Fanuc TP program (LS listing): S004.LS

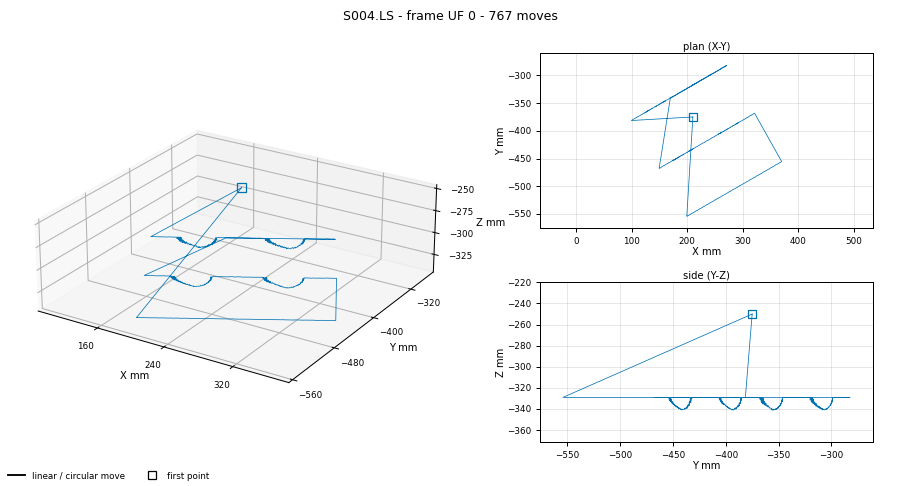
[picture p0: tool path of S004.LS in frame UF 0, 767 of 767 moves have a stored position in this frame; points joined in program order, loops and branches not executed]
/PROG  S004.LS
/ATTR
OWNER       = MNEDITOR;
COMMENT     = "";
PROG_SIZE   = 636;
CREATE      = DATE 23-01-07  TIME 11:59:14;
MODIFIED    = DATE 23-01-07  TIME 12:02:18;
FILE_NAME   = ;
VERSION     = 0;
LINE_COUNT  = 4;
MEMORY_SIZE = 992;
PROTECT     = READ_WRITE;
TCD:  STACK_SIZE	= 0,
      TASK_PRIORITY	= 50,
      TIME_SLICE	= 0,
      BUSY_LAMP_OFF	= 0,
      ABORT_REQUEST	= 0,
      PAUSE_REQUEST	= 0;
DEFAULT_GROUP	= 1,*,*,*,*;
CONTROL_CODE	= 00000000 00000000;
/MN
   1:J P[1] 100% FINE    ;
   2:L P[2] 100mm/sec CNT100    ;
   3:L P[3] 100mm/sec CNT100    ;
   4:L P[4] 100mm/sec CNT100    ;
   5:L P[5] 100mm/sec CNT100    ;
   6:L P[6] 100mm/sec CNT100    ;
   7:L P[7] 100mm/sec CNT100    ;
   8:L P[8] 100mm/sec CNT100    ;
   9:L P[9] 100mm/sec CNT100    ;
   10:L P[10] 100mm/sec CNT100    ;
   11:L P[11] 100mm/sec CNT100    ;
   12:L P[12] 100mm/sec CNT100    ;
   13:L P[13] 100mm/sec CNT100    ;
   14:L P[14] 100mm/sec CNT100    ;
   15:L P[15] 100mm/sec CNT100    ;
   16:L P[16] 100mm/sec CNT100    ;
   17:L P[17] 100mm/sec CNT100    ;
   18:L P[18] 100mm/sec CNT100    ;
   19:L P[19] 100mm/sec CNT100    ;
   20:L P[20] 100mm/sec CNT100    ;
   21:L P[21] 100mm/sec CNT100    ;
   22:L P[22] 100mm/sec CNT100    ;
   23:L P[23] 100mm/sec CNT100    ;
   24:L P[24] 100mm/sec CNT100    ;
   25:L P[25] 100mm/sec CNT100    ;
   26:L P[26] 100mm/sec CNT100    ;
   27:L P[27] 100mm/sec CNT100    ;
   28:L P[28] 100mm/sec CNT100    ;
   29:L P[29] 100mm/sec CNT100    ;
   30:L P[30] 100mm/sec CNT100    ;
   31:L P[31] 100mm/sec CNT100    ;
   32:L P[32] 100mm/sec CNT100    ;
   33:L P[33] 100mm/sec CNT100    ;
   34:L P[34] 100mm/sec CNT100    ;
   35:L P[35] 100mm/sec CNT100    ;
   36:L P[36] 100mm/sec CNT100    ;
   37:L P[37] 100mm/sec CNT100    ;
   38:L P[38] 100mm/sec CNT100    ;
   39:L P[39] 100mm/sec CNT100    ;
   40:L P[40] 100mm/sec CNT100    ;
   41:L P[41] 100mm/sec CNT100    ;
   42:L P[42] 100mm/sec CNT100    ;
   43:L P[43] 100mm/sec CNT100    ;
   44:L P[44] 100mm/sec CNT100    ;
   45:L P[45] 100mm/sec CNT100    ;
   46:L P[46] 100mm/sec CNT100    ;
   47:L P[47] 100mm/sec CNT100    ;
   48:L P[48] 100mm/sec CNT100    ;
   49:L P[49] 100mm/sec CNT100    ;
   50:L P[50] 100mm/sec CNT100    ;
   51:L P[51] 100mm/sec CNT100    ;
   52:L P[52] 100mm/sec CNT100    ;
   53:L P[53] 100mm/sec CNT100    ;
   54:L P[54] 100mm/sec CNT100    ;
   55:L P[55] 100mm/sec CNT100    ;
   56:L P[56] 100mm/sec CNT100    ;
   57:L P[57] 100mm/sec CNT100    ;
   58:L P[58] 100mm/sec CNT100    ;
   59:L P[59] 100mm/sec CNT100    ;
   60:L P[60] 100mm/sec CNT100    ;
   61:L P[61] 100mm/sec CNT100    ;
   62:L P[62] 100mm/sec CNT100    ;
   63:L P[63] 100mm/sec CNT100    ;
   64:L P[64] 100mm/sec CNT100    ;
   65:L P[65] 100mm/sec CNT100    ;
   66:L P[66] 100mm/sec CNT100    ;
   67:L P[67] 100mm/sec CNT100    ;
   68:L P[68] 100mm/sec CNT100    ;
   69:L P[69] 100mm/sec CNT100    ;
   70:L P[70] 100mm/sec CNT100    ;
   71:L P[71] 100mm/sec CNT100    ;
   72:L P[72] 100mm/sec CNT100    ;
   73:L P[73] 100mm/sec CNT100    ;
   74:L P[74] 100mm/sec CNT100    ;
   75:L P[75] 100mm/sec CNT100    ;
   76:L P[76] 100mm/sec CNT100    ;
   77:L P[77] 100mm/sec CNT100    ;
   78:L P[78] 100mm/sec CNT100    ;
   79:L P[79] 100mm/sec CNT100    ;
   80:L P[80] 100mm/sec CNT100    ;
   81:L P[81] 100mm/sec CNT100    ;
   82:L P[82] 100mm/sec CNT100    ;
   83:L P[83] 100mm/sec CNT100    ;
   84:L P[84] 100mm/sec CNT100    ;
   85:L P[85] 100mm/sec CNT100    ;
   86:L P[86] 100mm/sec CNT100    ;
   87:L P[87] 100mm/sec CNT100    ;
   88:L P[88] 100mm/sec CNT100    ;
   89:L P[89] 100mm/sec CNT100    ;
   90:L P[90] 100mm/sec CNT100    ;
   91:L P[91] 100mm/sec CNT100    ;
   92:L P[92] 100mm/sec CNT100    ;
   93:L P[93] 100mm/sec CNT100    ;
   94:L P[94] 100mm/sec CNT100    ;
   95:L P[95] 100mm/sec CNT100    ;
   96:L P[96] 100mm/sec CNT100    ;
   97:L P[97] 100mm/sec CNT100    ;
   98:L P[98] 100mm/sec CNT100    ;
   99:L P[99] 100mm/sec CNT100    ;
   100:L P[100] 100mm/sec CNT100    ;
   101:L P[101] 100mm/sec CNT100    ;
   102:L P[102] 100mm/sec CNT100    ;
   103:L P[103] 100mm/sec CNT100    ;
   104:L P[104] 100mm/sec CNT100    ;
   105:L P[105] 100mm/sec CNT100    ;
   106:L P[106] 100mm/sec CNT100    ;
   107:L P[107] 100mm/sec CNT100    ;
   108:L P[108] 100mm/sec CNT100    ;
   109:L P[109] 100mm/sec CNT100    ;
   110:L P[110] 100mm/sec CNT100    ;
   111:L P[111] 100mm/sec CNT100    ;
   112:L P[112] 100mm/sec CNT100    ;
   113:L P[113] 100mm/sec CNT100    ;
   114:L P[114] 100mm/sec CNT100    ;
   115:L P[115] 100mm/sec CNT100    ;
   116:L P[116] 100mm/sec CNT100    ;
   117:L P[117] 100mm/sec CNT100    ;
   118:L P[118] 100mm/sec CNT100    ;
   119:L P[119] 100mm/sec CNT100    ;
   120:L P[120] 100mm/sec CNT100    ;
   121:L P[121] 100mm/sec CNT100    ;
   122:L P[122] 100mm/sec CNT100    ;
   123:L P[123] 100mm/sec CNT100    ;
   124:L P[124] 100mm/sec CNT100    ;
   125:L P[125] 100mm/sec CNT100    ;
   126:L P[126] 100mm/sec CNT100    ;
   127:L P[127] 100mm/sec CNT100    ;
   128:L P[128] 100mm/sec CNT100    ;
   129:L P[129] 100mm/sec CNT100    ;
   130:L P[130] 100mm/sec CNT100    ;
   131:L P[131] 100mm/sec CNT100    ;
   132:L P[132] 100mm/sec CNT100    ;
   133:L P[133] 100mm/sec CNT100    ;
   134:L P[134] 100mm/sec CNT100    ;
   135:L P[135] 100mm/sec CNT100    ;
   136:L P[136] 100mm/sec CNT100    ;
   137:L P[137] 100mm/sec CNT100    ;
   138:L P[138] 100mm/sec CNT100    ;
   139:L P[139] 100mm/sec CNT100    ;
   140:L P[140] 100mm/sec CNT100    ;
   141:L P[141] 100mm/sec CNT100    ;
   142:L P[142] 100mm/sec CNT100    ;
   143:L P[143] 100mm/sec CNT100    ;
   144:L P[144] 100mm/sec CNT100    ;
   145:L P[145] 100mm/sec CNT100    ;
   146:L P[146] 100mm/sec CNT100    ;
   147:L P[147] 100mm/sec CNT100    ;
   148:L P[148] 100mm/sec CNT100    ;
   149:L P[149] 100mm/sec CNT100    ;
   150:L P[150] 100mm/sec CNT100    ;
   151:L P[151] 100mm/sec CNT100    ;
   152:L P[152] 100mm/sec CNT100    ;
   153:L P[153] 100mm/sec CNT100    ;
   154:L P[154] 100mm/sec CNT100    ;
   155:L P[155] 100mm/sec CNT100    ;
   156:L P[156] 100mm/sec CNT100    ;
   157:L P[157] 100mm/sec CNT100    ;
   158:L P[158] 100mm/sec CNT100    ;
   159:L P[159] 100mm/sec CNT100    ;
   160:L P[160] 100mm/sec CNT100    ;
   161:L P[161] 100mm/sec CNT100    ;
   162:L P[162] 100mm/sec CNT100    ;
   163:L P[163] 100mm/sec CNT100    ;
   164:L P[164] 100mm/sec CNT100    ;
   165:L P[165] 100mm/sec CNT100    ;
   166:L P[166] 100mm/sec CNT100    ;
   167:L P[167] 100mm/sec CNT100    ;
   168:L P[168] 100mm/sec CNT100    ;
   169:L P[169] 100mm/sec CNT100    ;
   170:L P[170] 100mm/sec CNT100    ;
   171:L P[171] 100mm/sec CNT100    ;
   172:L P[172] 100mm/sec CNT100    ;
   173:L P[173] 100mm/sec CNT100    ;
   174:L P[174] 100mm/sec CNT100    ;
   175:L P[175] 100mm/sec CNT100    ;
   176:L P[176] 100mm/sec CNT100    ;
   177:L P[177] 100mm/sec CNT100    ;
   178:L P[178] 100mm/sec CNT100    ;
   179:L P[179] 100mm/sec CNT100    ;
   180:L P[180] 100mm/sec CNT100    ;
   181:L P[181] 100mm/sec CNT100    ;
   182:L P[182] 100mm/sec CNT100    ;
   183:L P[183] 100mm/sec CNT100    ;
   184:L P[184] 100mm/sec CNT100    ;
   185:L P[185] 100mm/sec CNT100    ;
   186:L P[186] 100mm/sec CNT100    ;
   187:L P[187] 100mm/sec CNT100    ;
   188:L P[188] 100mm/sec CNT100    ;
   189:L P[189] 100mm/sec CNT100    ;
   190:L P[190] 100mm/sec CNT100    ;
   191:L P[191] 100mm/sec CNT100    ;
   192:L P[192] 100mm/sec CNT100    ;
   193:L P[193] 100mm/sec CNT100    ;
   194:L P[194] 100mm/sec CNT100    ;
   195:L P[195] 100mm/sec CNT100    ;
   196:L P[196] 100mm/sec CNT100    ;
   197:L P[197] 100mm/sec CNT100    ;
   198:L P[198] 100mm/sec CNT100    ;
   199:L P[199] 100mm/sec CNT100    ;
   200:L P[200] 100mm/sec CNT100    ;
   201:L P[201] 100mm/sec CNT100    ;
   202:L P[202] 100mm/sec CNT100    ;
   203:L P[203] 100mm/sec CNT100    ;
   204:L P[204] 100mm/sec CNT100    ;
   205:L P[205] 100mm/sec CNT100    ;
   206:L P[206] 100mm/sec CNT100    ;
   207:L P[207] 100mm/sec CNT100    ;
   208:L P[208] 100mm/sec CNT100    ;
   209:L P[209] 100mm/sec CNT100    ;
   210:L P[210] 100mm/sec CNT100    ;
   211:L P[211] 100mm/sec CNT100    ;
   212:L P[212] 100mm/sec CNT100    ;
   213:L P[213] 100mm/sec CNT100    ;
   214:L P[214] 100mm/sec CNT100    ;
   215:L P[215] 100mm/sec CNT100    ;
   216:L P[216] 100mm/sec CNT100    ;
   217:L P[217] 100mm/sec CNT100    ;
   218:L P[218] 100mm/sec CNT100    ;
   219:L P[219] 100mm/sec CNT100    ;
   220:L P[220] 100mm/sec CNT100    ;
   221:L P[221] 100mm/sec CNT100    ;
   222:L P[222] 100mm/sec CNT100    ;
   223:L P[223] 100mm/sec CNT100    ;
   224:L P[224] 100mm/sec CNT100    ;
   225:L P[225] 100mm/sec CNT100    ;
   226:L P[226] 100mm/sec CNT100    ;
   227:L P[227] 100mm/sec CNT100    ;
   228:L P[228] 100mm/sec CNT100    ;
   229:L P[229] 100mm/sec CNT100    ;
   230:L P[230] 100mm/sec CNT100    ;
   231:L P[231] 100mm/sec CNT100    ;
   232:L P[232] 100mm/sec CNT100    ;
   233:L P[233] 100mm/sec CNT100    ;
   234:L P[234] 100mm/sec CNT100    ;
   235:L P[235] 100mm/sec CNT100    ;
   236:L P[236] 100mm/sec CNT100    ;
   237:L P[237] 100mm/sec CNT100    ;
   238:L P[238] 100mm/sec CNT100    ;
   239:L P[239] 100mm/sec CNT100    ;
   240:L P[240] 100mm/sec CNT100    ;
   241:L P[241] 100mm/sec CNT100    ;
   242:L P[242] 100mm/sec CNT100    ;
   243:L P[243] 100mm/sec CNT100    ;
   244:L P[244] 100mm/sec CNT100    ;
   245:L P[245] 100mm/sec CNT100    ;
   246:L P[246] 100mm/sec CNT100    ;
   247:L P[247] 100mm/sec CNT100    ;
   248:L P[248] 100mm/sec CNT100    ;
   249:L P[249] 100mm/sec CNT100    ;
   250:L P[250] 100mm/sec CNT100    ;
   251:L P[251] 100mm/sec CNT100    ;
   252:L P[252] 100mm/sec CNT100    ;
   253:L P[253] 100mm/sec CNT100    ;
   254:L P[254] 100mm/sec CNT100    ;
   255:L P[255] 100mm/sec CNT100    ;
   256:L P[256] 100mm/sec CNT100    ;
   257:L P[257] 100mm/sec CNT100    ;
   258:L P[258] 100mm/sec CNT100    ;
   259:L P[259] 100mm/sec CNT100    ;
   260:L P[260] 100mm/sec CNT100    ;
   261:L P[261] 100mm/sec CNT100    ;
   262:L P[262] 100mm/sec CNT100    ;
   263:L P[263] 100mm/sec CNT100    ;
   264:L P[264] 100mm/sec CNT100    ;
   265:L P[265] 100mm/sec CNT100    ;
   266:L P[266] 100mm/sec CNT100    ;
   267:L P[267] 100mm/sec CNT100    ;
   268:L P[268] 100mm/sec CNT100    ;
   269:L P[269] 100mm/sec CNT100    ;
   270:L P[270] 100mm/sec CNT100    ;
   271:L P[271] 100mm/sec CNT100    ;
   272:L P[272] 100mm/sec CNT100    ;
   273:L P[273] 100mm/sec CNT100    ;
   274:L P[274] 100mm/sec CNT100    ;
   275:L P[275] 100mm/sec CNT100    ;
   276:L P[276] 100mm/sec CNT100    ;
   277:L P[277] 100mm/sec CNT100    ;
   278:L P[278] 100mm/sec CNT100    ;
   279:L P[279] 100mm/sec CNT100    ;
   280:L P[280] 100mm/sec CNT100    ;
   281:L P[281] 100mm/sec CNT100    ;
   282:L P[282] 100mm/sec CNT100    ;
   283:L P[283] 100mm/sec CNT100    ;
   284:L P[284] 100mm/sec CNT100    ;
   285:L P[285] 100mm/sec CNT100    ;
   286:L P[286] 100mm/sec CNT100    ;
   287:L P[287] 100mm/sec CNT100    ;
   288:L P[288] 100mm/sec CNT100    ;
   289:L P[289] 100mm/sec CNT100    ;
   290:L P[290] 100mm/sec CNT100    ;
   291:L P[291] 100mm/sec CNT100    ;
   292:L P[292] 100mm/sec CNT100    ;
   293:L P[293] 100mm/sec CNT100    ;
   294:L P[294] 100mm/sec CNT100    ;
   295:L P[295] 100mm/sec CNT100    ;
   296:L P[296] 100mm/sec CNT100    ;
   297:L P[297] 100mm/sec CNT100    ;
   298:L P[298] 100mm/sec CNT100    ;
   299:L P[299] 100mm/sec CNT100    ;
   300:L P[300] 100mm/sec CNT100    ;
   301:L P[301] 100mm/sec CNT100    ;
   302:L P[302] 100mm/sec CNT100    ;
   303:L P[303] 100mm/sec CNT100    ;
   304:L P[304] 100mm/sec CNT100    ;
   305:L P[305] 100mm/sec CNT100    ;
   306:L P[306] 100mm/sec CNT100    ;
   307:L P[307] 100mm/sec CNT100    ;
   308:L P[308] 100mm/sec CNT100    ;
   309:L P[309] 100mm/sec CNT100    ;
   310:L P[310] 100mm/sec CNT100    ;
   311:L P[311] 100mm/sec CNT100    ;
   312:L P[312] 100mm/sec CNT100    ;
   313:L P[313] 100mm/sec CNT100    ;
   314:L P[314] 100mm/sec CNT100    ;
   315:L P[315] 100mm/sec CNT100    ;
   316:L P[316] 100mm/sec CNT100    ;
   317:L P[317] 100mm/sec CNT100    ;
   318:L P[318] 100mm/sec CNT100    ;
   319:L P[319] 100mm/sec CNT100    ;
   320:L P[320] 100mm/sec CNT100    ;
   321:L P[321] 100mm/sec CNT100    ;
   322:L P[322] 100mm/sec CNT100    ;
   323:L P[323] 100mm/sec CNT100    ;
   324:L P[324] 100mm/sec CNT100    ;
   325:L P[325] 100mm/sec CNT100    ;
   326:L P[326] 100mm/sec CNT100    ;
   327:L P[327] 100mm/sec CNT100    ;
   328:L P[328] 100mm/sec CNT100    ;
   329:L P[329] 100mm/sec CNT100    ;
   330:L P[330] 100mm/sec CNT100    ;
   331:L P[331] 100mm/sec CNT100    ;
   332:L P[332] 100mm/sec CNT100    ;
   333:L P[333] 100mm/sec CNT100    ;
   334:L P[334] 100mm/sec CNT100    ;
   335:L P[335] 100mm/sec CNT100    ;
   336:L P[336] 100mm/sec CNT100    ;
   337:L P[337] 100mm/sec CNT100    ;
   338:L P[338] 100mm/sec CNT100    ;
   339:L P[339] 100mm/sec CNT100    ;
   340:L P[340] 100mm/sec CNT100    ;
   341:L P[341] 100mm/sec CNT100    ;
   342:L P[342] 100mm/sec CNT100    ;
   343:L P[343] 100mm/sec CNT100    ;
   344:L P[344] 100mm/sec CNT100    ;
   345:L P[345] 100mm/sec CNT100    ;
   346:L P[346] 100mm/sec CNT100    ;
   347:L P[347] 100mm/sec CNT100    ;
   348:L P[348] 100mm/sec CNT100    ;
   349:L P[349] 100mm/sec CNT100    ;
   350:L P[350] 100mm/sec CNT100    ;
   351:L P[351] 100mm/sec CNT100    ;
   352:L P[352] 100mm/sec CNT100    ;
   353:L P[353] 100mm/sec CNT100    ;
   354:L P[354] 100mm/sec CNT100    ;
   355:L P[355] 100mm/sec CNT100    ;
   356:L P[356] 100mm/sec CNT100    ;
   357:L P[357] 100mm/sec CNT100    ;
   358:L P[358] 100mm/sec CNT100    ;
   359:L P[359] 100mm/sec CNT100    ;
   360:L P[360] 100mm/sec CNT100    ;
   361:L P[361] 100mm/sec CNT100    ;
   362:L P[362] 100mm/sec CNT100    ;
   363:L P[363] 100mm/sec CNT100    ;
   364:L P[364] 100mm/sec CNT100    ;
   365:L P[365] 100mm/sec CNT100    ;
   366:L P[366] 100mm/sec CNT100    ;
   367:L P[367] 100mm/sec CNT100    ;
   368:L P[368] 100mm/sec CNT100    ;
   369:L P[369] 100mm/sec CNT100    ;
   370:L P[370] 100mm/sec CNT100    ;
   371:L P[371] 100mm/sec CNT100    ;
   372:L P[372] 100mm/sec CNT100    ;
   373:L P[373] 100mm/sec CNT100    ;
   374:L P[374] 100mm/sec CNT100    ;
   375:L P[375] 100mm/sec CNT100    ;
   376:L P[376] 100mm/sec CNT100    ;
   377:L P[377] 100mm/sec CNT100    ;
   378:L P[378] 100mm/sec CNT100    ;
   379:L P[379] 100mm/sec CNT100    ;
   380:L P[380] 100mm/sec CNT100    ;
   381:L P[381] 100mm/sec CNT100    ;
   382:L P[382] 100mm/sec CNT100    ;
   383:L P[383] 100mm/sec CNT100    ;
   384:L P[384] 100mm/sec CNT100    ;
   385:L P[385] 100mm/sec CNT100    ;
   386:L P[386] 100mm/sec CNT100    ;
   387:L P[387] 100mm/sec CNT100    ;
   388:L P[388] 100mm/sec CNT100    ;
   389:L P[389] 100mm/sec CNT100    ;
   390:L P[390] 100mm/sec CNT100    ;
   391:L P[391] 100mm/sec CNT100    ;
   392:L P[392] 100mm/sec CNT100    ;
   393:L P[393] 100mm/sec CNT100    ;
   394:L P[394] 100mm/sec CNT100    ;
   395:L P[395] 100mm/sec CNT100    ;
   396:L P[396] 100mm/sec CNT100    ;
   397:L P[397] 100mm/sec CNT100    ;
   398:L P[398] 100mm/sec CNT100    ;
   399:L P[399] 100mm/sec CNT100    ;
   400:L P[400] 100mm/sec CNT100    ;
   401:L P[401] 100mm/sec CNT100    ;
   402:L P[402] 100mm/sec CNT100    ;
   403:L P[403] 100mm/sec CNT100    ;
   404:L P[404] 100mm/sec CNT100    ;
   405:L P[405] 100mm/sec CNT100    ;
   406:L P[406] 100mm/sec CNT100    ;
   407:L P[407] 100mm/sec CNT100    ;
   408:L P[408] 100mm/sec CNT100    ;
   409:L P[409] 100mm/sec CNT100    ;
   410:L P[410] 100mm/sec CNT100    ;
   411:L P[411] 100mm/sec CNT100    ;
   412:L P[412] 100mm/sec CNT100    ;
   413:L P[413] 100mm/sec CNT100    ;
   414:L P[414] 100mm/sec CNT100    ;
   415:L P[415] 100mm/sec CNT100    ;
   416:L P[416] 100mm/sec CNT100    ;
   417:L P[417] 100mm/sec CNT100    ;
   418:L P[418] 100mm/sec CNT100    ;
   419:L P[419] 100mm/sec CNT100    ;
   420:L P[420] 100mm/sec CNT100    ;
   421:L P[421] 100mm/sec CNT100    ;
   422:L P[422] 100mm/sec CNT100    ;
   423:L P[423] 100mm/sec CNT100    ;
   424:L P[424] 100mm/sec CNT100    ;
   425:L P[425] 100mm/sec CNT100    ;
   426:L P[426] 100mm/sec CNT100    ;
   427:L P[427] 100mm/sec CNT100    ;
   428:L P[428] 100mm/sec CNT100    ;
   429:L P[429] 100mm/sec CNT100    ;
   430:L P[430] 100mm/sec CNT100    ;
   431:L P[431] 100mm/sec CNT100    ;
   432:L P[432] 100mm/sec CNT100    ;
   433:L P[433] 100mm/sec CNT100    ;
   434:L P[434] 100mm/sec CNT100    ;
   435:L P[435] 100mm/sec CNT100    ;
   436:L P[436] 100mm/sec CNT100    ;
   437:L P[437] 100mm/sec CNT100    ;
   438:L P[438] 100mm/sec CNT100    ;
   439:L P[439] 100mm/sec CNT100    ;
   440:L P[440] 100mm/sec CNT100    ;
   441:L P[441] 100mm/sec CNT100    ;
   442:L P[442] 100mm/sec CNT100    ;
   443:L P[443] 100mm/sec CNT100    ;
   444:L P[444] 100mm/sec CNT100    ;
   445:L P[445] 100mm/sec CNT100    ;
   446:L P[446] 100mm/sec CNT100    ;
   447:L P[447] 100mm/sec CNT100    ;
   448:L P[448] 100mm/sec CNT100    ;
   449:L P[449] 100mm/sec CNT100    ;
   450:L P[450] 100mm/sec CNT100    ;
   451:L P[451] 100mm/sec CNT100    ;
   452:L P[452] 100mm/sec CNT100    ;
   453:L P[453] 100mm/sec CNT100    ;
   454:L P[454] 100mm/sec CNT100    ;
   455:L P[455] 100mm/sec CNT100    ;
   456:L P[456] 100mm/sec CNT100    ;
   457:L P[457] 100mm/sec CNT100    ;
   458:L P[458] 100mm/sec CNT100    ;
   459:L P[459] 100mm/sec CNT100    ;
   460:L P[460] 100mm/sec CNT100    ;
   461:L P[461] 100mm/sec CNT100    ;
   462:L P[462] 100mm/sec CNT100    ;
   463:L P[463] 100mm/sec CNT100    ;
   464:L P[464] 100mm/sec CNT100    ;
   465:L P[465] 100mm/sec CNT100    ;
   466:L P[466] 100mm/sec CNT100    ;
   467:L P[467] 100mm/sec CNT100    ;
   468:L P[468] 100mm/sec CNT100    ;
   469:L P[469] 100mm/sec CNT100    ;
   470:L P[470] 100mm/sec CNT100    ;
   471:L P[471] 100mm/sec CNT100    ;
   472:L P[472] 100mm/sec CNT100    ;
   473:L P[473] 100mm/sec CNT100    ;
   474:L P[474] 100mm/sec CNT100    ;
   475:L P[475] 100mm/sec CNT100    ;
   476:L P[476] 100mm/sec CNT100    ;
   477:L P[477] 100mm/sec CNT100    ;
   478:L P[478] 100mm/sec CNT100    ;
   479:L P[479] 100mm/sec CNT100    ;
   480:L P[480] 100mm/sec CNT100    ;
   481:L P[481] 100mm/sec CNT100    ;
   482:L P[482] 100mm/sec CNT100    ;
   483:L P[483] 100mm/sec CNT100    ;
   484:L P[484] 100mm/sec CNT100    ;
   485:L P[485] 100mm/sec CNT100    ;
   486:L P[486] 100mm/sec CNT100    ;
   487:L P[487] 100mm/sec CNT100    ;
   488:L P[488] 100mm/sec CNT100    ;
   489:L P[489] 100mm/sec CNT100    ;
   490:L P[490] 100mm/sec CNT100    ;
   491:L P[491] 100mm/sec CNT100    ;
   492:L P[492] 100mm/sec CNT100    ;
   493:L P[493] 100mm/sec CNT100    ;
   494:L P[494] 100mm/sec CNT100    ;
   495:L P[495] 100mm/sec CNT100    ;
   496:L P[496] 100mm/sec CNT100    ;
   497:L P[497] 100mm/sec CNT100    ;
   498:L P[498] 100mm/sec CNT100    ;
   499:L P[499] 100mm/sec CNT100    ;
   500:L P[500] 100mm/sec CNT100    ;
   501:L P[501] 100mm/sec CNT100    ;
   502:L P[502] 100mm/sec CNT100    ;
   503:L P[503] 100mm/sec CNT100    ;
   504:L P[504] 100mm/sec CNT100    ;
   505:L P[505] 100mm/sec CNT100    ;
   506:L P[506] 100mm/sec CNT100    ;
   507:L P[507] 100mm/sec CNT100    ;
   508:L P[508] 100mm/sec CNT100    ;
   509:L P[509] 100mm/sec CNT100    ;
   510:L P[510] 100mm/sec CNT100    ;
   511:L P[511] 100mm/sec CNT100    ;
   512:L P[512] 100mm/sec CNT100    ;
   513:L P[513] 100mm/sec CNT100    ;
   514:L P[514] 100mm/sec CNT100    ;
   515:L P[515] 100mm/sec CNT100    ;
   516:L P[516] 100mm/sec CNT100    ;
   517:L P[517] 100mm/sec CNT100    ;
   518:L P[518] 100mm/sec CNT100    ;
   519:L P[519] 100mm/sec CNT100    ;
   520:L P[520] 100mm/sec CNT100    ;
   521:L P[521] 100mm/sec CNT100    ;
   522:L P[522] 100mm/sec CNT100    ;
   523:L P[523] 100mm/sec CNT100    ;
   524:L P[524] 100mm/sec CNT100    ;
   525:L P[525] 100mm/sec CNT100    ;
   526:L P[526] 100mm/sec CNT100    ;
   527:L P[527] 100mm/sec CNT100    ;
   528:L P[528] 100mm/sec CNT100    ;
   529:L P[529] 100mm/sec CNT100    ;
   530:L P[530] 100mm/sec CNT100    ;
   531:L P[531] 100mm/sec CNT100    ;
   532:L P[532] 100mm/sec CNT100    ;
   533:L P[533] 100mm/sec CNT100    ;
   534:L P[534] 100mm/sec CNT100    ;
   535:L P[535] 100mm/sec CNT100    ;
   536:L P[536] 100mm/sec CNT100    ;
   537:L P[537] 100mm/sec CNT100    ;
   538:L P[538] 100mm/sec CNT100    ;
   539:L P[539] 100mm/sec CNT100    ;
   540:L P[540] 100mm/sec CNT100    ;
   541:L P[541] 100mm/sec CNT100    ;
   542:L P[542] 100mm/sec CNT100    ;
   543:L P[543] 100mm/sec CNT100    ;
   544:L P[544] 100mm/sec CNT100    ;
   545:L P[545] 100mm/sec CNT100    ;
   546:L P[546] 100mm/sec CNT100    ;
   547:L P[547] 100mm/sec CNT100    ;
   548:L P[548] 100mm/sec CNT100    ;
   549:L P[549] 100mm/sec CNT100    ;
   550:L P[550] 100mm/sec CNT100    ;
   551:L P[551] 100mm/sec CNT100    ;
   552:L P[552] 100mm/sec CNT100    ;
   553:L P[553] 100mm/sec CNT100    ;
   554:L P[554] 100mm/sec CNT100    ;
   555:L P[555] 100mm/sec CNT100    ;
   556:L P[556] 100mm/sec CNT100    ;
   557:L P[557] 100mm/sec CNT100    ;
   558:L P[558] 100mm/sec CNT100    ;
   559:L P[559] 100mm/sec CNT100    ;
   560:L P[560] 100mm/sec CNT100    ;
   561:L P[561] 100mm/sec CNT100    ;
   562:L P[562] 100mm/sec CNT100    ;
   563:L P[563] 100mm/sec CNT100    ;
   564:L P[564] 100mm/sec CNT100    ;
   565:L P[565] 100mm/sec CNT100    ;
   566:L P[566] 100mm/sec CNT100    ;
   567:L P[567] 100mm/sec CNT100    ;
   568:L P[568] 100mm/sec CNT100    ;
   569:L P[569] 100mm/sec CNT100    ;
   570:L P[570] 100mm/sec CNT100    ;
   571:L P[571] 100mm/sec CNT100    ;
   572:L P[572] 100mm/sec CNT100    ;
   573:L P[573] 100mm/sec CNT100    ;
   574:L P[574] 100mm/sec CNT100    ;
   575:L P[575] 100mm/sec CNT100    ;
   576:L P[576] 100mm/sec CNT100    ;
   577:L P[577] 100mm/sec CNT100    ;
   578:L P[578] 100mm/sec CNT100    ;
   579:L P[579] 100mm/sec CNT100    ;
   580:L P[580] 100mm/sec CNT100    ;
   581:L P[581] 100mm/sec CNT100    ;
   582:L P[582] 100mm/sec CNT100    ;
   583:L P[583] 100mm/sec CNT100    ;
   584:L P[584] 100mm/sec CNT100    ;
   585:L P[585] 100mm/sec CNT100    ;
   586:L P[586] 100mm/sec CNT100    ;
   587:L P[587] 100mm/sec CNT100    ;
   588:L P[588] 100mm/sec CNT100    ;
   589:L P[589] 100mm/sec CNT100    ;
   590:L P[590] 100mm/sec CNT100    ;
   591:L P[591] 100mm/sec CNT100    ;
   592:L P[592] 100mm/sec CNT100    ;
   593:L P[593] 100mm/sec CNT100    ;
   594:L P[594] 100mm/sec CNT100    ;
   595:L P[595] 100mm/sec CNT100    ;
   596:L P[596] 100mm/sec CNT100    ;
   597:L P[597] 100mm/sec CNT100    ;
   598:L P[598] 100mm/sec CNT100    ;
   599:L P[599] 100mm/sec CNT100    ;
   600:L P[600] 100mm/sec CNT100    ;
   601:L P[601] 100mm/sec CNT100    ;
   602:L P[602] 100mm/sec CNT100    ;
   603:L P[603] 100mm/sec CNT100    ;
   604:L P[604] 100mm/sec CNT100    ;
   605:L P[605] 100mm/sec CNT100    ;
   606:L P[606] 100mm/sec CNT100    ;
   607:L P[607] 100mm/sec CNT100    ;
   608:L P[608] 100mm/sec CNT100    ;
   609:L P[609] 100mm/sec CNT100    ;
   610:L P[610] 100mm/sec CNT100    ;
   611:L P[611] 100mm/sec CNT100    ;
   612:L P[612] 100mm/sec CNT100    ;
   613:L P[613] 100mm/sec CNT100    ;
   614:L P[614] 100mm/sec CNT100    ;
   615:L P[615] 100mm/sec CNT100    ;
   616:L P[616] 100mm/sec CNT100    ;
   617:L P[617] 100mm/sec CNT100    ;
   618:L P[618] 100mm/sec CNT100    ;
   619:L P[619] 100mm/sec CNT100    ;
   620:L P[620] 100mm/sec CNT100    ;
   621:L P[621] 100mm/sec CNT100    ;
   622:L P[622] 100mm/sec CNT100    ;
   623:L P[623] 100mm/sec CNT100    ;
   624:L P[624] 100mm/sec CNT100    ;
   625:L P[625] 100mm/sec CNT100    ;
   626:L P[626] 100mm/sec CNT100    ;
   627:L P[627] 100mm/sec CNT100    ;
   628:L P[628] 100mm/sec CNT100    ;
   629:L P[629] 100mm/sec CNT100    ;
   630:L P[630] 100mm/sec CNT100    ;
   631:L P[631] 100mm/sec CNT100    ;
   632:L P[632] 100mm/sec CNT100    ;
   633:L P[633] 100mm/sec CNT100    ;
   634:L P[634] 100mm/sec CNT100    ;
   635:L P[635] 100mm/sec CNT100    ;
   636:L P[636] 100mm/sec CNT100    ;
   637:L P[637] 100mm/sec CNT100    ;
   638:L P[638] 100mm/sec CNT100    ;
   639:L P[639] 100mm/sec CNT100    ;
   640:L P[640] 100mm/sec CNT100    ;
   641:L P[641] 100mm/sec CNT100    ;
   642:L P[642] 100mm/sec CNT100    ;
   643:L P[643] 100mm/sec CNT100    ;
   644:L P[644] 100mm/sec CNT100    ;
   645:L P[645] 100mm/sec CNT100    ;
   646:L P[646] 100mm/sec CNT100    ;
   647:L P[647] 100mm/sec CNT100    ;
   648:L P[648] 100mm/sec CNT100    ;
   649:L P[649] 100mm/sec CNT100    ;
   650:L P[650] 100mm/sec CNT100    ;
   651:L P[651] 100mm/sec CNT100    ;
   652:L P[652] 100mm/sec CNT100    ;
   653:L P[653] 100mm/sec CNT100    ;
   654:L P[654] 100mm/sec CNT100    ;
   655:L P[655] 100mm/sec CNT100    ;
   656:L P[656] 100mm/sec CNT100    ;
   657:L P[657] 100mm/sec CNT100    ;
   658:L P[658] 100mm/sec CNT100    ;
   659:L P[659] 100mm/sec CNT100    ;
   660:L P[660] 100mm/sec CNT100    ;
   661:L P[661] 100mm/sec CNT100    ;
   662:L P[662] 100mm/sec CNT100    ;
   663:L P[663] 100mm/sec CNT100    ;
   664:L P[664] 100mm/sec CNT100    ;
   665:L P[665] 100mm/sec CNT100    ;
   666:L P[666] 100mm/sec CNT100    ;
   667:L P[667] 100mm/sec CNT100    ;
   668:L P[668] 100mm/sec CNT100    ;
   669:L P[669] 100mm/sec CNT100    ;
   670:L P[670] 100mm/sec CNT100    ;
   671:L P[671] 100mm/sec CNT100    ;
   672:L P[672] 100mm/sec CNT100    ;
   673:L P[673] 100mm/sec CNT100    ;
   674:L P[674] 100mm/sec CNT100    ;
   675:L P[675] 100mm/sec CNT100    ;
   676:L P[676] 100mm/sec CNT100    ;
   677:L P[677] 100mm/sec CNT100    ;
   678:L P[678] 100mm/sec CNT100    ;
   679:L P[679] 100mm/sec CNT100    ;
   680:L P[680] 100mm/sec CNT100    ;
   681:L P[681] 100mm/sec CNT100    ;
   682:L P[682] 100mm/sec CNT100    ;
   683:L P[683] 100mm/sec CNT100    ;
   684:L P[684] 100mm/sec CNT100    ;
   685:L P[685] 100mm/sec CNT100    ;
   686:L P[686] 100mm/sec CNT100    ;
   687:L P[687] 100mm/sec CNT100    ;
   688:L P[688] 100mm/sec CNT100    ;
   689:L P[689] 100mm/sec CNT100    ;
   690:L P[690] 100mm/sec CNT100    ;
   691:L P[691] 100mm/sec CNT100    ;
   692:L P[692] 100mm/sec CNT100    ;
   693:L P[693] 100mm/sec CNT100    ;
   694:L P[694] 100mm/sec CNT100    ;
   695:L P[695] 100mm/sec CNT100    ;
   696:L P[696] 100mm/sec CNT100    ;
   697:L P[697] 100mm/sec CNT100    ;
   698:L P[698] 100mm/sec CNT100    ;
   699:L P[699] 100mm/sec CNT100    ;
   700:L P[700] 100mm/sec CNT100    ;
   701:L P[701] 100mm/sec CNT100    ;
   702:L P[702] 100mm/sec CNT100    ;
   703:L P[703] 100mm/sec CNT100    ;
   704:L P[704] 100mm/sec CNT100    ;
   705:L P[705] 100mm/sec CNT100    ;
   706:L P[706] 100mm/sec CNT100    ;
   707:L P[707] 100mm/sec CNT100    ;
   708:L P[708] 100mm/sec CNT100    ;
   709:L P[709] 100mm/sec CNT100    ;
   710:L P[710] 100mm/sec CNT100    ;
   711:L P[711] 100mm/sec CNT100    ;
   712:L P[712] 100mm/sec CNT100    ;
   713:L P[713] 100mm/sec CNT100    ;
   714:L P[714] 100mm/sec CNT100    ;
   715:L P[715] 100mm/sec CNT100    ;
   716:L P[716] 100mm/sec CNT100    ;
   717:L P[717] 100mm/sec CNT100    ;
   718:L P[718] 100mm/sec CNT100    ;
   719:L P[719] 100mm/sec CNT100    ;
   720:L P[720] 100mm/sec CNT100    ;
   721:L P[721] 100mm/sec CNT100    ;
   722:L P[722] 100mm/sec CNT100    ;
   723:L P[723] 100mm/sec CNT100    ;
   724:L P[724] 100mm/sec CNT100    ;
   725:L P[725] 100mm/sec CNT100    ;
   726:L P[726] 100mm/sec CNT100    ;
   727:L P[727] 100mm/sec CNT100    ;
   728:L P[728] 100mm/sec CNT100    ;
   729:L P[729] 100mm/sec CNT100    ;
   730:L P[730] 100mm/sec CNT100    ;
   731:L P[731] 100mm/sec CNT100    ;
   732:L P[732] 100mm/sec CNT100    ;
   733:L P[733] 100mm/sec CNT100    ;
   734:L P[734] 100mm/sec CNT100    ;
   735:L P[735] 100mm/sec CNT100    ;
   736:L P[736] 100mm/sec CNT100    ;
   737:L P[737] 100mm/sec CNT100    ;
   738:L P[738] 100mm/sec CNT100    ;
   739:L P[739] 100mm/sec CNT100    ;
   740:L P[740] 100mm/sec CNT100    ;
   741:L P[741] 100mm/sec CNT100    ;
   742:L P[742] 100mm/sec CNT100    ;
   743:L P[743] 100mm/sec CNT100    ;
   744:L P[744] 100mm/sec CNT100    ;
   745:L P[745] 100mm/sec CNT100    ;
   746:L P[746] 100mm/sec CNT100    ;
   747:L P[747] 100mm/sec CNT100    ;
   748:L P[748] 100mm/sec CNT100    ;
   749:L P[749] 100mm/sec CNT100    ;
   750:L P[750] 100mm/sec CNT100    ;
   751:L P[751] 100mm/sec CNT100    ;
   752:L P[752] 100mm/sec CNT100    ;
   753:L P[753] 100mm/sec CNT100    ;
   754:L P[754] 100mm/sec CNT100    ;
   755:L P[755] 100mm/sec CNT100    ;
   756:L P[756] 100mm/sec CNT100    ;
   757:L P[757] 100mm/sec CNT100    ;
   758:L P[758] 100mm/sec CNT100    ;
   759:L P[759] 100mm/sec CNT100    ;
   760:L P[760] 100mm/sec CNT100    ;
   761:L P[761] 100mm/sec CNT100    ;
   762:L P[762] 100mm/sec CNT100    ;
   763:L P[763] 100mm/sec CNT100    ;
   764:L P[764] 100mm/sec CNT100    ;
   765:L P[765] 100mm/sec CNT100    ;
   766:L P[766] 100mm/sec CNT100    ;
   767:L P[767] 100mm/sec CNT100    ;
/POS
P[1]{
   GP1:
	UF : 0, UT : 6,		CONFIG : 'N U T, 0, 0, 0',
	X =  210.000  mm,	Y =   -375.000  mm,	Z =   -250.000  mm,
	W =  90.000 deg,	P =   0.000 deg,	R =   90.000 deg
};
P[2]{
   GP1:
	UF : 0, UT : 6,		CONFIG : 'N U T, 0, 0, 0',
	X =  99.048  mm,	Y =   -381.442  mm,	Z =   -329.000  mm,
	W =  90.000 deg,	P =   0.000 deg,	R =   90.000 deg
};
P[3]{
   GP1:
	UF : 0, UT : 6,		CONFIG : 'N U T, 0, 0, 0',
	X =  99.873  mm,	Y =   -380.917  mm,	Z =   -329.000  mm,
	W =  90.000 deg,	P =   0.000 deg,	R =   90.000 deg
};
P[4]{
   GP1:
	UF : 0, UT : 6,		CONFIG : 'N U T, 0, 0, 0',
	X =  100.888  mm,	Y =   -380.459  mm,	Z =   -329.000  mm,
	W =  90.000 deg,	P =   0.000 deg,	R =   90.000 deg
};
P[5]{
   GP1:
	UF : 0, UT : 6,		CONFIG : 'N U T, 0, 0, 0',
	X =  101.765  mm,	Y =   -379.889  mm,	Z =   -329.000  mm,
	W =  90.000 deg,	P =   0.000 deg,	R =   90.000 deg
};
P[6]{
   GP1:
	UF : 0, UT : 6,		CONFIG : 'N U T, 0, 0, 0',
	X =  102.835  mm,	Y =   -379.243  mm,	Z =   -329.000  mm,
	W =  90.000 deg,	P =   0.000 deg,	R =   90.000 deg
};
P[7]{
   GP1:
	UF : 0, UT : 6,		CONFIG : 'N U T, 0, 0, 0',
	X =  103.446  mm,	Y =   -378.703  mm,	Z =   -329.000  mm,
	W =  90.000 deg,	P =   0.000 deg,	R =   90.000 deg
};
P[8]{
   GP1:
	UF : 0, UT : 6,		CONFIG : 'N U T, 0, 0, 0',
	X =  104.720  mm,	Y =   -378.117  mm,	Z =   -329.100  mm,
	W =  90.000 deg,	P =   0.000 deg,	R =   90.000 deg
};
P[9]{
   GP1:
	UF : 0, UT : 6,		CONFIG : 'N U T, 0, 0, 0',
	X =  105.487  mm,	Y =   -377.698  mm,	Z =   -329.100  mm,
	W =  90.000 deg,	P =   0.000 deg,	R =   90.000 deg
};
P[10]{
   GP1:
	UF : 0, UT : 6,		CONFIG : 'N U T, 0, 0, 0',
	X =  106.013  mm,	Y =   -376.984  mm,	Z =   -329.100  mm,
	W =  90.000 deg,	P =   0.000 deg,	R =   90.000 deg
};
P[11]{
   GP1:
	UF : 0, UT : 6,		CONFIG : 'N U T, 0, 0, 0',
	X =  107.136  mm,	Y =   -376.661  mm,	Z =   -329.100  mm,
	W =  90.000 deg,	P =   0.000 deg,	R =   90.000 deg
};
P[12]{
   GP1:
	UF : 0, UT : 6,		CONFIG : 'N U T, 0, 0, 0',
	X =  108.278  mm,	Y =   -376.323  mm,	Z =   -329.100  mm,
	W =  90.000 deg,	P =   0.000 deg,	R =   90.000 deg
};
P[13]{
   GP1:
	UF : 0, UT : 6,		CONFIG : 'N U T, 0, 0, 0',
	X =  108.277  mm,	Y =   -375.570  mm,	Z =   -329.100  mm,
	W =  90.000 deg,	P =   0.000 deg,	R =   90.000 deg
};
P[14]{
   GP1:
	UF : 0, UT : 6,		CONFIG : 'N U T, 0, 0, 0',
	X =  109.543  mm,	Y =   -375.332  mm,	Z =   -329.100  mm,
	W =  90.000 deg,	P =   0.000 deg,	R =   90.000 deg
};
P[15]{
   GP1:
	UF : 0, UT : 6,		CONFIG : 'N U T, 0, 0, 0',
	X =  110.173  mm,	Y =   -374.706  mm,	Z =   -329.100  mm,
	W =  90.000 deg,	P =   0.000 deg,	R =   90.000 deg
};
P[16]{
   GP1:
	UF : 0, UT : 6,		CONFIG : 'N U T, 0, 0, 0',
	X =  111.478  mm,	Y =   -374.378  mm,	Z =   -329.100  mm,
	W =  90.000 deg,	P =   0.000 deg,	R =   90.000 deg
};
P[17]{
   GP1:
	UF : 0, UT : 6,		CONFIG : 'N U T, 0, 0, 0',
	X =  112.258  mm,	Y =   -373.714  mm,	Z =   -329.100  mm,
	W =  90.000 deg,	P =   0.000 deg,	R =   90.000 deg
};
P[18]{
   GP1:
	UF : 0, UT : 6,		CONFIG : 'N U T, 0, 0, 0',
	X =  113.122  mm,	Y =   -373.332  mm,	Z =   -329.100  mm,
	W =  90.000 deg,	P =   0.000 deg,	R =   90.000 deg
};
P[19]{
   GP1:
	UF : 0, UT : 6,		CONFIG : 'N U T, 0, 0, 0',
	X =  113.794  mm,	Y =   -372.981  mm,	Z =   -329.100  mm,
	W =  90.000 deg,	P =   0.000 deg,	R =   90.000 deg
};
P[20]{
   GP1:
	UF : 0, UT : 6,		CONFIG : 'N U T, 0, 0, 0',
	X =  114.977  mm,	Y =   -372.274  mm,	Z =   -329.100  mm,
	W =  90.000 deg,	P =   0.000 deg,	R =   90.000 deg
};
P[21]{
   GP1:
	UF : 0, UT : 6,		CONFIG : 'N U T, 0, 0, 0',
	X =  116.486  mm,	Y =   -370.959  mm,	Z =   -329.100  mm,
	W =  90.000 deg,	P =   0.000 deg,	R =   90.000 deg
};
P[22]{
   GP1:
	UF : 0, UT : 6,		CONFIG : 'N U T, 0, 0, 0',
	X =  117.328  mm,	Y =   -370.667  mm,	Z =   -329.100  mm,
	W =  90.000 deg,	P =   0.000 deg,	R =   90.000 deg
};
P[23]{
   GP1:
	UF : 0, UT : 6,		CONFIG : 'N U T, 0, 0, 0',
	X =  118.060  mm,	Y =   -370.578  mm,	Z =   -329.100  mm,
	W =  90.000 deg,	P =   0.000 deg,	R =   90.000 deg
};
P[24]{
   GP1:
	UF : 0, UT : 6,		CONFIG : 'N U T, 0, 0, 0',
	X =  118.805  mm,	Y =   -369.926  mm,	Z =   -329.100  mm,
	W =  90.000 deg,	P =   0.000 deg,	R =   90.000 deg
};
P[25]{
   GP1:
	UF : 0, UT : 6,		CONFIG : 'N U T, 0, 0, 0',
	X =  121.351  mm,	Y =   -368.870  mm,	Z =   -329.100  mm,
	W =  90.000 deg,	P =   0.000 deg,	R =   90.000 deg
};
P[26]{
   GP1:
	UF : 0, UT : 6,		CONFIG : 'N U T, 0, 0, 0',
	X =  121.913  mm,	Y =   -368.223  mm,	Z =   -329.100  mm,
	W =  90.000 deg,	P =   0.000 deg,	R =   90.000 deg
};
P[27]{
   GP1:
	UF : 0, UT : 6,		CONFIG : 'N U T, 0, 0, 0',
	X =  122.724  mm,	Y =   -367.614  mm,	Z =   -329.100  mm,
	W =  90.000 deg,	P =   0.000 deg,	R =   90.000 deg
};
P[28]{
   GP1:
	UF : 0, UT : 6,		CONFIG : 'N U T, 0, 0, 0',
	X =  122.976  mm,	Y =   -368.036  mm,	Z =   -329.794  mm,
	W =  90.000 deg,	P =   0.000 deg,	R =   90.000 deg
};
P[29]{
   GP1:
	UF : 0, UT : 6,		CONFIG : 'N U T, 0, 0, 0',
	X =  123.638  mm,	Y =   -367.486  mm,	Z =   -329.858  mm,
	W =  90.000 deg,	P =   0.000 deg,	R =   90.000 deg
};
P[30]{
   GP1:
	UF : 0, UT : 6,		CONFIG : 'N U T, 0, 0, 0',
	X =  123.861  mm,	Y =   -367.444  mm,	Z =   -331.084  mm,
	W =  90.000 deg,	P =   0.000 deg,	R =   90.000 deg
};
P[31]{
   GP1:
	UF : 0, UT : 6,		CONFIG : 'N U T, 0, 0, 0',
	X =  123.786  mm,	Y =   -366.752  mm,	Z =   -329.100  mm,
	W =  90.000 deg,	P =   0.000 deg,	R =   90.000 deg
};
P[32]{
   GP1:
	UF : 0, UT : 6,		CONFIG : 'N U T, 0, 0, 0',
	X =  124.228  mm,	Y =   -367.081  mm,	Z =   -330.632  mm,
	W =  90.000 deg,	P =   0.000 deg,	R =   90.000 deg
};
P[33]{
   GP1:
	UF : 0, UT : 6,		CONFIG : 'N U T, 0, 0, 0',
	X =  124.388  mm,	Y =   -366.328  mm,	Z =   -329.100  mm,
	W =  90.000 deg,	P =   0.000 deg,	R =   90.000 deg
};
P[34]{
   GP1:
	UF : 0, UT : 6,		CONFIG : 'N U T, 0, 0, 0',
	X =  124.726  mm,	Y =   -366.578  mm,	Z =   -329.906  mm,
	W =  90.000 deg,	P =   0.000 deg,	R =   90.000 deg
};
P[35]{
   GP1:
	UF : 0, UT : 6,		CONFIG : 'N U T, 0, 0, 0',
	X =  124.826  mm,	Y =   -366.694  mm,	Z =   -331.608  mm,
	W =  90.000 deg,	P =   0.000 deg,	R =   90.000 deg
};
P[36]{
   GP1:
	UF : 0, UT : 6,		CONFIG : 'N U T, 0, 0, 0',
	X =  125.309  mm,	Y =   -366.449  mm,	Z =   -332.180  mm,
	W =  90.000 deg,	P =   0.000 deg,	R =   90.000 deg
};
P[37]{
   GP1:
	UF : 0, UT : 6,		CONFIG : 'N U T, 0, 0, 0',
	X =  125.324  mm,	Y =   -366.183  mm,	Z =   -330.835  mm,
	W =  90.000 deg,	P =   0.000 deg,	R =   90.000 deg
};
P[38]{
   GP1:
	UF : 0, UT : 6,		CONFIG : 'N U T, 0, 0, 0',
	X =  125.416  mm,	Y =   -365.999  mm,	Z =   -329.905  mm,
	W =  90.000 deg,	P =   0.000 deg,	R =   90.000 deg
};
P[39]{
   GP1:
	UF : 0, UT : 6,		CONFIG : 'N U T, 0, 0, 0',
	X =  125.864  mm,	Y =   -366.416  mm,	Z =   -333.461  mm,
	W =  90.000 deg,	P =   0.000 deg,	R =   90.000 deg
};
P[40]{
   GP1:
	UF : 0, UT : 6,		CONFIG : 'N U T, 0, 0, 0',
	X =  125.983  mm,	Y =   -365.959  mm,	Z =   -332.452  mm,
	W =  90.000 deg,	P =   0.000 deg,	R =   90.000 deg
};
P[41]{
   GP1:
	UF : 0, UT : 6,		CONFIG : 'N U T, 0, 0, 0',
	X =  126.005  mm,	Y =   -365.673  mm,	Z =   -331.367  mm,
	W =  90.000 deg,	P =   0.000 deg,	R =   90.000 deg
};
P[42]{
   GP1:
	UF : 0, UT : 6,		CONFIG : 'N U T, 0, 0, 0',
	X =  126.084  mm,	Y =   -365.207  mm,	Z =   -329.100  mm,
	W =  90.000 deg,	P =   0.000 deg,	R =   90.000 deg
};
P[43]{
   GP1:
	UF : 0, UT : 6,		CONFIG : 'N U T, 0, 0, 0',
	X =  126.601  mm,	Y =   -365.966  mm,	Z =   -333.948  mm,
	W =  90.000 deg,	P =   0.000 deg,	R =   90.000 deg
};
P[44]{
   GP1:
	UF : 0, UT : 6,		CONFIG : 'N U T, 0, 0, 0',
	X =  126.541  mm,	Y =   -365.718  mm,	Z =   -333.135  mm,
	W =  90.000 deg,	P =   0.000 deg,	R =   90.000 deg
};
P[45]{
   GP1:
	UF : 0, UT : 6,		CONFIG : 'N U T, 0, 0, 0',
	X =  126.298  mm,	Y =   -365.277  mm,	Z =   -330.098  mm,
	W =  90.000 deg,	P =   0.000 deg,	R =   90.000 deg
};
P[46]{
   GP1:
	UF : 0, UT : 6,		CONFIG : 'N U T, 0, 0, 0',
	X =  126.867  mm,	Y =   -364.890  mm,	Z =   -330.884  mm,
	W =  90.000 deg,	P =   0.000 deg,	R =   90.000 deg
};
P[47]{
   GP1:
	UF : 0, UT : 6,		CONFIG : 'N U T, 0, 0, 0',
	X =  127.182  mm,	Y =   -365.368  mm,	Z =   -333.669  mm,
	W =  90.000 deg,	P =   0.000 deg,	R =   90.000 deg
};
P[48]{
   GP1:
	UF : 0, UT : 6,		CONFIG : 'N U T, 0, 0, 0',
	X =  126.978  mm,	Y =   -364.963  mm,	Z =   -331.902  mm,
	W =  90.000 deg,	P =   0.000 deg,	R =   90.000 deg
};
P[49]{
   GP1:
	UF : 0, UT : 6,		CONFIG : 'N U T, 0, 0, 0',
	X =  127.187  mm,	Y =   -364.509  mm,	Z =   -329.860  mm,
	W =  90.000 deg,	P =   0.000 deg,	R =   90.000 deg
};
P[50]{
   GP1:
	UF : 0, UT : 6,		CONFIG : 'N U T, 0, 0, 0',
	X =  127.559  mm,	Y =   -364.554  mm,	Z =   -332.197  mm,
	W =  90.000 deg,	P =   0.000 deg,	R =   90.000 deg
};
P[51]{
   GP1:
	UF : 0, UT : 6,		CONFIG : 'N U T, 0, 0, 0',
	X =  127.779  mm,	Y =   -364.665  mm,	Z =   -333.143  mm,
	W =  90.000 deg,	P =   0.000 deg,	R =   90.000 deg
};
P[52]{
   GP1:
	UF : 0, UT : 6,		CONFIG : 'N U T, 0, 0, 0',
	X =  127.630  mm,	Y =   -364.274  mm,	Z =   -331.104  mm,
	W =  90.000 deg,	P =   0.000 deg,	R =   90.000 deg
};
P[53]{
   GP1:
	UF : 0, UT : 6,		CONFIG : 'N U T, 0, 0, 0',
	X =  128.324  mm,	Y =   -364.991  mm,	Z =   -334.995  mm,
	W =  90.000 deg,	P =   0.000 deg,	R =   90.000 deg
};
P[54]{
   GP1:
	UF : 0, UT : 6,		CONFIG : 'N U T, 0, 0, 0',
	X =  128.319  mm,	Y =   -364.514  mm,	Z =   -333.986  mm,
	W =  90.000 deg,	P =   0.000 deg,	R =   90.000 deg
};
P[55]{
   GP1:
	UF : 0, UT : 6,		CONFIG : 'N U T, 0, 0, 0',
	X =  128.319  mm,	Y =   -364.133  mm,	Z =   -332.946  mm,
	W =  90.000 deg,	P =   0.000 deg,	R =   90.000 deg
};
P[56]{
   GP1:
	UF : 0, UT : 6,		CONFIG : 'N U T, 0, 0, 0',
	X =  129.109  mm,	Y =   -364.506  mm,	Z =   -335.364  mm,
	W =  90.000 deg,	P =   0.000 deg,	R =   90.000 deg
};
P[57]{
   GP1:
	UF : 0, UT : 6,		CONFIG : 'N U T, 0, 0, 0',
	X =  128.767  mm,	Y =   -363.632  mm,	Z =   -332.534  mm,
	W =  90.000 deg,	P =   0.000 deg,	R =   90.000 deg
};
P[58]{
   GP1:
	UF : 0, UT : 6,		CONFIG : 'N U T, 0, 0, 0',
	X =  129.474  mm,	Y =   -363.428  mm,	Z =   -333.711  mm,
	W =  90.000 deg,	P =   0.000 deg,	R =   90.000 deg
};
P[59]{
   GP1:
	UF : 0, UT : 6,		CONFIG : 'N U T, 0, 0, 0',
	X =  129.757  mm,	Y =   -363.830  mm,	Z =   -335.129  mm,
	W =  90.000 deg,	P =   0.000 deg,	R =   90.000 deg
};
P[60]{
   GP1:
	UF : 0, UT : 6,		CONFIG : 'N U T, 0, 0, 0',
	X =  130.207  mm,	Y =   -363.348  mm,	Z =   -334.942  mm,
	W =  90.000 deg,	P =   0.000 deg,	R =   90.000 deg
};
P[61]{
   GP1:
	UF : 0, UT : 6,		CONFIG : 'N U T, 0, 0, 0',
	X =  130.414  mm,	Y =   -362.748  mm,	Z =   -334.047  mm,
	W =  90.000 deg,	P =   0.000 deg,	R =   90.000 deg
};
P[62]{
   GP1:
	UF : 0, UT : 6,		CONFIG : 'N U T, 0, 0, 0',
	X =  130.910  mm,	Y =   -363.387  mm,	Z =   -336.096  mm,
	W =  90.000 deg,	P =   0.000 deg,	R =   90.000 deg
};
P[63]{
   GP1:
	UF : 0, UT : 6,		CONFIG : 'N U T, 0, 0, 0',
	X =  131.169  mm,	Y =   -362.680  mm,	Z =   -335.251  mm,
	W =  90.000 deg,	P =   0.000 deg,	R =   90.000 deg
};
P[64]{
   GP1:
	UF : 0, UT : 6,		CONFIG : 'N U T, 0, 0, 0',
	X =  131.898  mm,	Y =   -362.755  mm,	Z =   -336.459  mm,
	W =  90.000 deg,	P =   0.000 deg,	R =   90.000 deg
};
P[65]{
   GP1:
	UF : 0, UT : 6,		CONFIG : 'N U T, 0, 0, 0',
	X =  131.947  mm,	Y =   -362.309  mm,	Z =   -335.834  mm,
	W =  90.000 deg,	P =   0.000 deg,	R =   90.000 deg
};
P[66]{
   GP1:
	UF : 0, UT : 6,		CONFIG : 'N U T, 0, 0, 0',
	X =  131.812  mm,	Y =   -361.883  mm,	Z =   -334.768  mm,
	W =  90.000 deg,	P =   0.000 deg,	R =   90.000 deg
};
P[67]{
   GP1:
	UF : 0, UT : 6,		CONFIG : 'N U T, 0, 0, 0',
	X =  132.642  mm,	Y =   -361.583  mm,	Z =   -335.582  mm,
	W =  90.000 deg,	P =   0.000 deg,	R =   90.000 deg
};
P[68]{
   GP1:
	UF : 0, UT : 6,		CONFIG : 'N U T, 0, 0, 0',
	X =  133.031  mm,	Y =   -361.959  mm,	Z =   -336.760  mm,
	W =  90.000 deg,	P =   0.000 deg,	R =   90.000 deg
};
P[69]{
   GP1:
	UF : 0, UT : 6,		CONFIG : 'N U T, 0, 0, 0',
	X =  133.676  mm,	Y =   -361.545  mm,	Z =   -336.973  mm,
	W =  90.000 deg,	P =   0.000 deg,	R =   90.000 deg
};
P[70]{
   GP1:
	UF : 0, UT : 6,		CONFIG : 'N U T, 0, 0, 0',
	X =  133.814  mm,	Y =   -361.032  mm,	Z =   -336.390  mm,
	W =  90.000 deg,	P =   0.000 deg,	R =   90.000 deg
};
P[71]{
   GP1:
	UF : 0, UT : 6,		CONFIG : 'N U T, 0, 0, 0',
	X =  135.194  mm,	Y =   -360.791  mm,	Z =   -337.749  mm,
	W =  90.000 deg,	P =   0.000 deg,	R =   90.000 deg
};
P[72]{
   GP1:
	UF : 0, UT : 6,		CONFIG : 'N U T, 0, 0, 0',
	X =  135.362  mm,	Y =   -359.951  mm,	Z =   -336.817  mm,
	W =  90.000 deg,	P =   0.000 deg,	R =   90.000 deg
};
P[73]{
   GP1:
	UF : 0, UT : 6,		CONFIG : 'N U T, 0, 0, 0',
	X =  135.760  mm,	Y =   -360.228  mm,	Z =   -337.663  mm,
	W =  90.000 deg,	P =   0.000 deg,	R =   90.000 deg
};
P[74]{
   GP1:
	UF : 0, UT : 6,		CONFIG : 'N U T, 0, 0, 0',
	X =  136.452  mm,	Y =   -359.868  mm,	Z =   -337.996  mm,
	W =  90.000 deg,	P =   0.000 deg,	R =   90.000 deg
};
P[75]{
   GP1:
	UF : 0, UT : 6,		CONFIG : 'N U T, 0, 0, 0',
	X =  136.276  mm,	Y =   -359.481  mm,	Z =   -337.278  mm,
	W =  90.000 deg,	P =   0.000 deg,	R =   90.000 deg
};
P[76]{
   GP1:
	UF : 0, UT : 6,		CONFIG : 'N U T, 0, 0, 0',
	X =  137.047  mm,	Y =   -359.425  mm,	Z =   -338.104  mm,
	W =  90.000 deg,	P =   0.000 deg,	R =   90.000 deg
};
P[77]{
   GP1:
	UF : 0, UT : 6,		CONFIG : 'N U T, 0, 0, 0',
	X =  138.067  mm,	Y =   -358.563  mm,	Z =   -338.156  mm,
	W =  90.000 deg,	P =   0.000 deg,	R =   90.000 deg
};
P[78]{
   GP1:
	UF : 0, UT : 6,		CONFIG : 'N U T, 0, 0, 0',
	X =  138.478  mm,	Y =   -358.817  mm,	Z =   -338.971  mm,
	W =  90.000 deg,	P =   0.000 deg,	R =   90.000 deg
};
P[79]{
   GP1:
	UF : 0, UT : 6,		CONFIG : 'N U T, 0, 0, 0',
	X =  139.210  mm,	Y =   -358.310  mm,	Z =   -339.103  mm,
	W =  90.000 deg,	P =   0.000 deg,	R =   90.000 deg
};
P[80]{
   GP1:
	UF : 0, UT : 6,		CONFIG : 'N U T, 0, 0, 0',
	X =  140.033  mm,	Y =   -357.554  mm,	Z =   -339.093  mm,
	W =  90.000 deg,	P =   0.000 deg,	R =   90.000 deg
};
P[81]{
   GP1:
	UF : 0, UT : 6,		CONFIG : 'N U T, 0, 0, 0',
	X =  140.897  mm,	Y =   -356.967  mm,	Z =   -339.350  mm,
	W =  90.000 deg,	P =   0.000 deg,	R =   90.000 deg
};
P[82]{
   GP1:
	UF : 0, UT : 6,		CONFIG : 'N U T, 0, 0, 0',
	X =  141.512  mm,	Y =   -356.346  mm,	Z =   -339.245  mm,
	W =  90.000 deg,	P =   0.000 deg,	R =   90.000 deg
};
P[83]{
   GP1:
	UF : 0, UT : 6,		CONFIG : 'N U T, 0, 0, 0',
	X =  141.986  mm,	Y =   -357.006  mm,	Z =   -340.349  mm,
	W =  90.000 deg,	P =   0.000 deg,	R =   90.000 deg
};
P[84]{
   GP1:
	UF : 0, UT : 6,		CONFIG : 'N U T, 0, 0, 0',
	X =  142.522  mm,	Y =   -356.284  mm,	Z =   -340.133  mm,
	W =  90.000 deg,	P =   0.000 deg,	R =   90.000 deg
};
P[85]{
   GP1:
	UF : 0, UT : 6,		CONFIG : 'N U T, 0, 0, 0',
	X =  143.044  mm,	Y =   -356.390  mm,	Z =   -340.689  mm,
	W =  90.000 deg,	P =   0.000 deg,	R =   90.000 deg
};
P[86]{
   GP1:
	UF : 0, UT : 6,		CONFIG : 'N U T, 0, 0, 0',
	X =  143.391  mm,	Y =   -355.717  mm,	Z =   -340.354  mm,
	W =  90.000 deg,	P =   0.000 deg,	R =   90.000 deg
};
P[87]{
   GP1:
	UF : 0, UT : 6,		CONFIG : 'N U T, 0, 0, 0',
	X =  143.714  mm,	Y =   -356.052  mm,	Z =   -340.952  mm,
	W =  90.000 deg,	P =   0.000 deg,	R =   90.000 deg
};
P[88]{
   GP1:
	UF : 0, UT : 6,		CONFIG : 'N U T, 0, 0, 0',
	X =  143.689  mm,	Y =   -355.108  mm,	Z =   -340.037  mm,
	W =  90.000 deg,	P =   0.000 deg,	R =   90.000 deg
};
P[89]{
   GP1:
	UF : 0, UT : 6,		CONFIG : 'N U T, 0, 0, 0',
	X =  144.518  mm,	Y =   -355.428  mm,	Z =   -341.062  mm,
	W =  90.000 deg,	P =   0.000 deg,	R =   90.000 deg
};
P[90]{
   GP1:
	UF : 0, UT : 6,		CONFIG : 'N U T, 0, 0, 0',
	X =  144.676  mm,	Y =   -354.636  mm,	Z =   -340.355  mm,
	W =  90.000 deg,	P =   0.000 deg,	R =   90.000 deg
};
P[91]{
   GP1:
	UF : 0, UT : 6,		CONFIG : 'N U T, 0, 0, 0',
	X =  145.198  mm,	Y =   -354.895  mm,	Z =   -340.929  mm,
	W =  90.000 deg,	P =   0.000 deg,	R =   90.000 deg
};
P[92]{
   GP1:
	UF : 0, UT : 6,		CONFIG : 'N U T, 0, 0, 0',
	X =  145.737  mm,	Y =   -354.267  mm,	Z =   -340.502  mm,
	W =  90.000 deg,	P =   0.000 deg,	R =   90.000 deg
};
P[93]{
   GP1:
	UF : 0, UT : 6,		CONFIG : 'N U T, 0, 0, 0',
	X =  146.889  mm,	Y =   -353.648  mm,	Z =   -340.413  mm,
	W =  90.000 deg,	P =   0.000 deg,	R =   90.000 deg
};
P[94]{
   GP1:
	UF : 0, UT : 6,		CONFIG : 'N U T, 0, 0, 0',
	X =  147.325  mm,	Y =   -353.018  mm,	Z =   -339.926  mm,
	W =  90.000 deg,	P =   0.000 deg,	R =   90.000 deg
};
P[95]{
   GP1:
	UF : 0, UT : 6,		CONFIG : 'N U T, 0, 0, 0',
	X =  147.898  mm,	Y =   -353.546  mm,	Z =   -340.834  mm,
	W =  90.000 deg,	P =   0.000 deg,	R =   90.000 deg
};
P[96]{
   GP1:
	UF : 0, UT : 6,		CONFIG : 'N U T, 0, 0, 0',
	X =  148.570  mm,	Y =   -352.459  mm,	Z =   -339.873  mm,
	W =  90.000 deg,	P =   0.000 deg,	R =   90.000 deg
};
P[97]{
   GP1:
	UF : 0, UT : 6,		CONFIG : 'N U T, 0, 0, 0',
	X =  149.600  mm,	Y =   -352.396  mm,	Z =   -340.210  mm,
	W =  90.000 deg,	P =   0.000 deg,	R =   90.000 deg
};
P[98]{
   GP1:
	UF : 0, UT : 6,		CONFIG : 'N U T, 0, 0, 0',
	X =  149.455  mm,	Y =   -351.803  mm,	Z =   -339.395  mm,
	W =  90.000 deg,	P =   0.000 deg,	R =   90.000 deg
};
P[99]{
   GP1:
	UF : 0, UT : 6,		CONFIG : 'N U T, 0, 0, 0',
	X =  150.390  mm,	Y =   -351.528  mm,	Z =   -339.470  mm,
	W =  90.000 deg,	P =   0.000 deg,	R =   90.000 deg
};
P[100]{
   GP1:
	UF : 0, UT : 6,		CONFIG : 'N U T, 0, 0, 0',
	X =  150.820  mm,	Y =   -351.979  mm,	Z =   -340.192  mm,
	W =  90.000 deg,	P =   0.000 deg,	R =   90.000 deg
};
P[101]{
   GP1:
	UF : 0, UT : 6,		CONFIG : 'N U T, 0, 0, 0',
	X =  151.161  mm,	Y =   -351.092  mm,	Z =   -339.183  mm,
	W =  90.000 deg,	P =   0.000 deg,	R =   90.000 deg
};
P[102]{
   GP1:
	UF : 0, UT : 6,		CONFIG : 'N U T, 0, 0, 0',
	X =  151.532  mm,	Y =   -350.516  mm,	Z =   -338.467  mm,
	W =  90.000 deg,	P =   0.000 deg,	R =   90.000 deg
};
P[103]{
   GP1:
	UF : 0, UT : 6,		CONFIG : 'N U T, 0, 0, 0',
	X =  152.019  mm,	Y =   -351.310  mm,	Z =   -339.858  mm,
	W =  90.000 deg,	P =   0.000 deg,	R =   90.000 deg
};
P[104]{
   GP1:
	UF : 0, UT : 6,		CONFIG : 'N U T, 0, 0, 0',
	X =  152.231  mm,	Y =   -350.557  mm,	Z =   -338.842  mm,
	W =  90.000 deg,	P =   0.000 deg,	R =   90.000 deg
};
P[105]{
   GP1:
	UF : 0, UT : 6,		CONFIG : 'N U T, 0, 0, 0',
	X =  152.395  mm,	Y =   -350.085  mm,	Z =   -338.078  mm,
	W =  90.000 deg,	P =   0.000 deg,	R =   90.000 deg
};
P[106]{
   GP1:
	UF : 0, UT : 6,		CONFIG : 'N U T, 0, 0, 0',
	X =  152.875  mm,	Y =   -349.680  mm,	Z =   -337.565  mm,
	W =  90.000 deg,	P =   0.000 deg,	R =   90.000 deg
};
P[107]{
   GP1:
	UF : 0, UT : 6,		CONFIG : 'N U T, 0, 0, 0',
	X =  153.392  mm,	Y =   -350.457  mm,	Z =   -339.123  mm,
	W =  90.000 deg,	P =   0.000 deg,	R =   90.000 deg
};
P[108]{
   GP1:
	UF : 0, UT : 6,		CONFIG : 'N U T, 0, 0, 0',
	X =  153.952  mm,	Y =   -349.700  mm,	Z =   -338.044  mm,
	W =  90.000 deg,	P =   0.000 deg,	R =   90.000 deg
};
P[109]{
   GP1:
	UF : 0, UT : 6,		CONFIG : 'N U T, 0, 0, 0',
	X =  154.082  mm,	Y =   -349.052  mm,	Z =   -336.956  mm,
	W =  90.000 deg,	P =   0.000 deg,	R =   90.000 deg
};
P[110]{
   GP1:
	UF : 0, UT : 6,		CONFIG : 'N U T, 0, 0, 0',
	X =  155.115  mm,	Y =   -349.185  mm,	Z =   -337.615  mm,
	W =  90.000 deg,	P =   0.000 deg,	R =   90.000 deg
};
P[111]{
   GP1:
	UF : 0, UT : 6,		CONFIG : 'N U T, 0, 0, 0',
	X =  155.097  mm,	Y =   -348.830  mm,	Z =   -336.984  mm,
	W =  90.000 deg,	P =   0.000 deg,	R =   90.000 deg
};
P[112]{
   GP1:
	UF : 0, UT : 6,		CONFIG : 'N U T, 0, 0, 0',
	X =  155.723  mm,	Y =   -348.299  mm,	Z =   -336.079  mm,
	W =  90.000 deg,	P =   0.000 deg,	R =   90.000 deg
};
P[113]{
   GP1:
	UF : 0, UT : 6,		CONFIG : 'N U T, 0, 0, 0',
	X =  156.082  mm,	Y =   -347.942  mm,	Z =   -335.260  mm,
	W =  90.000 deg,	P =   0.000 deg,	R =   90.000 deg
};
P[114]{
   GP1:
	UF : 0, UT : 6,		CONFIG : 'N U T, 0, 0, 0',
	X =  156.563  mm,	Y =   -348.658  mm,	Z =   -337.044  mm,
	W =  90.000 deg,	P =   0.000 deg,	R =   90.000 deg
};
P[115]{
   GP1:
	UF : 0, UT : 6,		CONFIG : 'N U T, 0, 0, 0',
	X =  156.550  mm,	Y =   -348.097  mm,	Z =   -335.868  mm,
	W =  90.000 deg,	P =   0.000 deg,	R =   90.000 deg
};
P[116]{
   GP1:
	UF : 0, UT : 6,		CONFIG : 'N U T, 0, 0, 0',
	X =  156.708  mm,	Y =   -347.682  mm,	Z =   -334.811  mm,
	W =  90.000 deg,	P =   0.000 deg,	R =   90.000 deg
};
P[117]{
   GP1:
	UF : 0, UT : 6,		CONFIG : 'N U T, 0, 0, 0',
	X =  157.439  mm,	Y =   -348.043  mm,	Z =   -336.085  mm,
	W =  90.000 deg,	P =   0.000 deg,	R =   90.000 deg
};
P[118]{
   GP1:
	UF : 0, UT : 6,		CONFIG : 'N U T, 0, 0, 0',
	X =  157.427  mm,	Y =   -347.394  mm,	Z =   -334.323  mm,
	W =  90.000 deg,	P =   0.000 deg,	R =   90.000 deg
};
P[119]{
   GP1:
	UF : 0, UT : 6,		CONFIG : 'N U T, 0, 0, 0',
	X =  157.460  mm,	Y =   -347.076  mm,	Z =   -333.224  mm,
	W =  90.000 deg,	P =   0.000 deg,	R =   90.000 deg
};
P[120]{
   GP1:
	UF : 0, UT : 6,		CONFIG : 'N U T, 0, 0, 0',
	X =  158.098  mm,	Y =   -347.522  mm,	Z =   -334.943  mm,
	W =  90.000 deg,	P =   0.000 deg,	R =   90.000 deg
};
P[121]{
   GP1:
	UF : 0, UT : 6,		CONFIG : 'N U T, 0, 0, 0',
	X =  158.312  mm,	Y =   -346.756  mm,	Z =   -332.401  mm,
	W =  90.000 deg,	P =   0.000 deg,	R =   90.000 deg
};
P[122]{
   GP1:
	UF : 0, UT : 6,		CONFIG : 'N U T, 0, 0, 0',
	X =  158.503  mm,	Y =   -346.945  mm,	Z =   -333.418  mm,
	W =  90.000 deg,	P =   0.000 deg,	R =   90.000 deg
};
P[123]{
   GP1:
	UF : 0, UT : 6,		CONFIG : 'N U T, 0, 0, 0',
	X =  158.648  mm,	Y =   -347.141  mm,	Z =   -334.134  mm,
	W =  90.000 deg,	P =   0.000 deg,	R =   90.000 deg
};
P[124]{
   GP1:
	UF : 0, UT : 6,		CONFIG : 'N U T, 0, 0, 0',
	X =  158.949  mm,	Y =   -346.756  mm,	Z =   -332.771  mm,
	W =  90.000 deg,	P =   0.000 deg,	R =   90.000 deg
};
P[125]{
   GP1:
	UF : 0, UT : 6,		CONFIG : 'N U T, 0, 0, 0',
	X =  158.864  mm,	Y =   -346.454  mm,	Z =   -330.983  mm,
	W =  90.000 deg,	P =   0.000 deg,	R =   90.000 deg
};
P[126]{
   GP1:
	UF : 0, UT : 6,		CONFIG : 'N U T, 0, 0, 0',
	X =  159.471  mm,	Y =   -346.992  mm,	Z =   -333.891  mm,
	W =  90.000 deg,	P =   0.000 deg,	R =   90.000 deg
};
P[127]{
   GP1:
	UF : 0, UT : 6,		CONFIG : 'N U T, 0, 0, 0',
	X =  159.164  mm,	Y =   -346.379  mm,	Z =   -330.247  mm,
	W =  90.000 deg,	P =   0.000 deg,	R =   90.000 deg
};
P[128]{
   GP1:
	UF : 0, UT : 6,		CONFIG : 'N U T, 0, 0, 0',
	X =  159.937  mm,	Y =   -346.692  mm,	Z =   -332.784  mm,
	W =  90.000 deg,	P =   0.000 deg,	R =   90.000 deg
};
P[129]{
   GP1:
	UF : 0, UT : 6,		CONFIG : 'N U T, 0, 0, 0',
	X =  159.660  mm,	Y =   -346.172  mm,	Z =   -329.100  mm,
	W =  90.000 deg,	P =   0.000 deg,	R =   90.000 deg
};
P[130]{
   GP1:
	UF : 0, UT : 6,		CONFIG : 'N U T, 0, 0, 0',
	X =  159.986  mm,	Y =   -346.382  mm,	Z =   -331.225  mm,
	W =  90.000 deg,	P =   0.000 deg,	R =   90.000 deg
};
P[131]{
   GP1:
	UF : 0, UT : 6,		CONFIG : 'N U T, 0, 0, 0',
	X =  159.975  mm,	Y =   -346.303  mm,	Z =   -330.051  mm,
	W =  90.000 deg,	P =   0.000 deg,	R =   90.000 deg
};
P[132]{
   GP1:
	UF : 0, UT : 6,		CONFIG : 'N U T, 0, 0, 0',
	X =  160.662  mm,	Y =   -346.297  mm,	Z =   -330.751  mm,
	W =  90.000 deg,	P =   0.000 deg,	R =   90.000 deg
};
P[133]{
   GP1:
	UF : 0, UT : 6,		CONFIG : 'N U T, 0, 0, 0',
	X =  160.759  mm,	Y =   -346.232  mm,	Z =   -329.900  mm,
	W =  90.000 deg,	P =   0.000 deg,	R =   90.000 deg
};
P[134]{
   GP1:
	UF : 0, UT : 6,		CONFIG : 'N U T, 0, 0, 0',
	X =  160.700  mm,	Y =   -345.963  mm,	Z =   -329.100  mm,
	W =  90.000 deg,	P =   0.000 deg,	R =   90.000 deg
};
P[135]{
   GP1:
	UF : 0, UT : 6,		CONFIG : 'N U T, 0, 0, 0',
	X =  161.089  mm,	Y =   -345.279  mm,	Z =   -329.100  mm,
	W =  90.000 deg,	P =   0.000 deg,	R =   90.000 deg
};
P[136]{
   GP1:
	UF : 0, UT : 6,		CONFIG : 'N U T, 0, 0, 0',
	X =  162.690  mm,	Y =   -344.677  mm,	Z =   -329.100  mm,
	W =  90.000 deg,	P =   0.000 deg,	R =   90.000 deg
};
P[137]{
   GP1:
	UF : 0, UT : 6,		CONFIG : 'N U T, 0, 0, 0',
	X =  163.171  mm,	Y =   -344.227  mm,	Z =   -329.100  mm,
	W =  90.000 deg,	P =   0.000 deg,	R =   90.000 deg
};
P[138]{
   GP1:
	UF : 0, UT : 6,		CONFIG : 'N U T, 0, 0, 0',
	X =  163.993  mm,	Y =   -343.609  mm,	Z =   -329.100  mm,
	W =  90.000 deg,	P =   0.000 deg,	R =   90.000 deg
};
P[139]{
   GP1:
	UF : 0, UT : 6,		CONFIG : 'N U T, 0, 0, 0',
	X =  165.385  mm,	Y =   -342.931  mm,	Z =   -329.100  mm,
	W =  90.000 deg,	P =   0.000 deg,	R =   90.000 deg
};
P[140]{
   GP1:
	UF : 0, UT : 6,		CONFIG : 'N U T, 0, 0, 0',
	X =  166.954  mm,	Y =   -342.281  mm,	Z =   -329.100  mm,
	W =  90.000 deg,	P =   0.000 deg,	R =   90.000 deg
};
P[141]{
   GP1:
	UF : 0, UT : 6,		CONFIG : 'N U T, 0, 0, 0',
	X =  167.835  mm,	Y =   -341.452  mm,	Z =   -329.100  mm,
	W =  90.000 deg,	P =   0.000 deg,	R =   90.000 deg
};
P[142]{
   GP1:
	UF : 0, UT : 6,		CONFIG : 'N U T, 0, 0, 0',
	X =  168.373  mm,	Y =   -340.740  mm,	Z =   -329.100  mm,
	W =  90.000 deg,	P =   0.000 deg,	R =   90.000 deg
};
P[143]{
   GP1:
	UF : 0, UT : 6,		CONFIG : 'N U T, 0, 0, 0',
	X =  170.533  mm,	Y =   -339.967  mm,	Z =   -329.100  mm,
	W =  90.000 deg,	P =   0.000 deg,	R =   90.000 deg
};
P[144]{
   GP1:
	UF : 0, UT : 6,		CONFIG : 'N U T, 0, 0, 0',
	X =  171.181  mm,	Y =   -339.251  mm,	Z =   -329.100  mm,
	W =  90.000 deg,	P =   0.000 deg,	R =   90.000 deg
};
P[145]{
   GP1:
	UF : 0, UT : 6,		CONFIG : 'N U T, 0, 0, 0',
	X =  171.860  mm,	Y =   -338.791  mm,	Z =   -329.100  mm,
	W =  90.000 deg,	P =   0.000 deg,	R =   90.000 deg
};
P[146]{
   GP1:
	UF : 0, UT : 6,		CONFIG : 'N U T, 0, 0, 0',
	X =  172.669  mm,	Y =   -338.935  mm,	Z =   -329.100  mm,
	W =  90.000 deg,	P =   0.000 deg,	R =   90.000 deg
};
P[147]{
   GP1:
	UF : 0, UT : 6,		CONFIG : 'N U T, 0, 0, 0',
	X =  173.432  mm,	Y =   -338.262  mm,	Z =   -329.100  mm,
	W =  90.000 deg,	P =   0.000 deg,	R =   90.000 deg
};
P[148]{
   GP1:
	UF : 0, UT : 6,		CONFIG : 'N U T, 0, 0, 0',
	X =  174.647  mm,	Y =   -337.719  mm,	Z =   -329.100  mm,
	W =  90.000 deg,	P =   0.000 deg,	R =   90.000 deg
};
P[149]{
   GP1:
	UF : 0, UT : 6,		CONFIG : 'N U T, 0, 0, 0',
	X =  176.046  mm,	Y =   -336.881  mm,	Z =   -329.000  mm,
	W =  90.000 deg,	P =   0.000 deg,	R =   90.000 deg
};
P[150]{
   GP1:
	UF : 0, UT : 6,		CONFIG : 'N U T, 0, 0, 0',
	X =  176.771  mm,	Y =   -336.215  mm,	Z =   -329.000  mm,
	W =  90.000 deg,	P =   0.000 deg,	R =   90.000 deg
};
P[151]{
   GP1:
	UF : 0, UT : 6,		CONFIG : 'N U T, 0, 0, 0',
	X =  178.042  mm,	Y =   -335.986  mm,	Z =   -329.000  mm,
	W =  90.000 deg,	P =   0.000 deg,	R =   90.000 deg
};
P[152]{
   GP1:
	UF : 0, UT : 6,		CONFIG : 'N U T, 0, 0, 0',
	X =  178.749  mm,	Y =   -335.521  mm,	Z =   -329.000  mm,
	W =  90.000 deg,	P =   0.000 deg,	R =   90.000 deg
};
P[153]{
   GP1:
	UF : 0, UT : 6,		CONFIG : 'N U T, 0, 0, 0',
	X =  180.628  mm,	Y =   -334.149  mm,	Z =   -329.000  mm,
	W =  90.000 deg,	P =   0.000 deg,	R =   90.000 deg
};
P[154]{
   GP1:
	UF : 0, UT : 6,		CONFIG : 'N U T, 0, 0, 0',
	X =  181.570  mm,	Y =   -333.551  mm,	Z =   -329.000  mm,
	W =  90.000 deg,	P =   0.000 deg,	R =   90.000 deg
};
P[155]{
   GP1:
	UF : 0, UT : 6,		CONFIG : 'N U T, 0, 0, 0',
	X =  182.242  mm,	Y =   -333.236  mm,	Z =   -329.000  mm,
	W =  90.000 deg,	P =   0.000 deg,	R =   90.000 deg
};
P[156]{
   GP1:
	UF : 0, UT : 6,		CONFIG : 'N U T, 0, 0, 0',
	X =  183.370  mm,	Y =   -332.730  mm,	Z =   -329.000  mm,
	W =  90.000 deg,	P =   0.000 deg,	R =   90.000 deg
};
P[157]{
   GP1:
	UF : 0, UT : 6,		CONFIG : 'N U T, 0, 0, 0',
	X =  184.284  mm,	Y =   -331.877  mm,	Z =   -329.000  mm,
	W =  90.000 deg,	P =   0.000 deg,	R =   90.000 deg
};
P[158]{
   GP1:
	UF : 0, UT : 6,		CONFIG : 'N U T, 0, 0, 0',
	X =  185.798  mm,	Y =   -331.270  mm,	Z =   -329.000  mm,
	W =  90.000 deg,	P =   0.000 deg,	R =   90.000 deg
};
P[159]{
   GP1:
	UF : 0, UT : 6,		CONFIG : 'N U T, 0, 0, 0',
	X =  186.804  mm,	Y =   -330.775  mm,	Z =   -329.050  mm,
	W =  90.000 deg,	P =   0.000 deg,	R =   90.000 deg
};
P[160]{
   GP1:
	UF : 0, UT : 6,		CONFIG : 'N U T, 0, 0, 0',
	X =  187.853  mm,	Y =   -330.379  mm,	Z =   -329.100  mm,
	W =  90.000 deg,	P =   0.000 deg,	R =   90.000 deg
};
P[161]{
   GP1:
	UF : 0, UT : 6,		CONFIG : 'N U T, 0, 0, 0',
	X =  188.465  mm,	Y =   -329.658  mm,	Z =   -329.100  mm,
	W =  90.000 deg,	P =   0.000 deg,	R =   90.000 deg
};
P[162]{
   GP1:
	UF : 0, UT : 6,		CONFIG : 'N U T, 0, 0, 0',
	X =  188.795  mm,	Y =   -329.004  mm,	Z =   -329.100  mm,
	W =  90.000 deg,	P =   0.000 deg,	R =   90.000 deg
};
P[163]{
   GP1:
	UF : 0, UT : 6,		CONFIG : 'N U T, 0, 0, 0',
	X =  189.691  mm,	Y =   -328.704  mm,	Z =   -329.100  mm,
	W =  90.000 deg,	P =   0.000 deg,	R =   90.000 deg
};
P[164]{
   GP1:
	UF : 0, UT : 6,		CONFIG : 'N U T, 0, 0, 0',
	X =  190.868  mm,	Y =   -328.375  mm,	Z =   -329.100  mm,
	W =  90.000 deg,	P =   0.000 deg,	R =   90.000 deg
};
P[165]{
   GP1:
	UF : 0, UT : 6,		CONFIG : 'N U T, 0, 0, 0',
	X =  192.216  mm,	Y =   -327.729  mm,	Z =   -329.100  mm,
	W =  90.000 deg,	P =   0.000 deg,	R =   90.000 deg
};
P[166]{
   GP1:
	UF : 0, UT : 6,		CONFIG : 'N U T, 0, 0, 0',
	X =  192.982  mm,	Y =   -327.042  mm,	Z =   -329.100  mm,
	W =  90.000 deg,	P =   0.000 deg,	R =   90.000 deg
};
P[167]{
   GP1:
	UF : 0, UT : 6,		CONFIG : 'N U T, 0, 0, 0',
	X =  193.958  mm,	Y =   -326.470  mm,	Z =   -329.100  mm,
	W =  90.000 deg,	P =   0.000 deg,	R =   90.000 deg
};
P[168]{
   GP1:
	UF : 0, UT : 6,		CONFIG : 'N U T, 0, 0, 0',
	X =  194.722  mm,	Y =   -326.462  mm,	Z =   -329.100  mm,
	W =  90.000 deg,	P =   0.000 deg,	R =   90.000 deg
};
P[169]{
   GP1:
	UF : 0, UT : 6,		CONFIG : 'N U T, 0, 0, 0',
	X =  195.615  mm,	Y =   -325.762  mm,	Z =   -329.100  mm,
	W =  90.000 deg,	P =   0.000 deg,	R =   90.000 deg
};
P[170]{
   GP1:
	UF : 0, UT : 6,		CONFIG : 'N U T, 0, 0, 0',
	X =  196.248  mm,	Y =   -325.018  mm,	Z =   -329.100  mm,
	W =  90.000 deg,	P =   0.000 deg,	R =   90.000 deg
};
P[171]{
   GP1:
	UF : 0, UT : 6,		CONFIG : 'N U T, 0, 0, 0',
	X =  197.107  mm,	Y =   -325.019  mm,	Z =   -329.100  mm,
	W =  90.000 deg,	P =   0.000 deg,	R =   90.000 deg
};
P[172]{
   GP1:
	UF : 0, UT : 6,		CONFIG : 'N U T, 0, 0, 0',
	X =  198.289  mm,	Y =   -324.378  mm,	Z =   -329.100  mm,
	W =  90.000 deg,	P =   0.000 deg,	R =   90.000 deg
};
P[173]{
   GP1:
	UF : 0, UT : 6,		CONFIG : 'N U T, 0, 0, 0',
	X =  199.019  mm,	Y =   -323.730  mm,	Z =   -329.100  mm,
	W =  90.000 deg,	P =   0.000 deg,	R =   90.000 deg
};
P[174]{
   GP1:
	UF : 0, UT : 6,		CONFIG : 'N U T, 0, 0, 0',
	X =  199.698  mm,	Y =   -322.692  mm,	Z =   -329.100  mm,
	W =  90.000 deg,	P =   0.000 deg,	R =   90.000 deg
};
P[175]{
   GP1:
	UF : 0, UT : 6,		CONFIG : 'N U T, 0, 0, 0',
	X =  200.649  mm,	Y =   -322.319  mm,	Z =   -329.100  mm,
	W =  90.000 deg,	P =   0.000 deg,	R =   90.000 deg
};
P[176]{
   GP1:
	UF : 0, UT : 6,		CONFIG : 'N U T, 0, 0, 0',
	X =  201.860  mm,	Y =   -322.287  mm,	Z =   -329.100  mm,
	W =  90.000 deg,	P =   0.000 deg,	R =   90.000 deg
};
P[177]{
   GP1:
	UF : 0, UT : 6,		CONFIG : 'N U T, 0, 0, 0',
	X =  202.148  mm,	Y =   -321.539  mm,	Z =   -329.100  mm,
	W =  90.000 deg,	P =   0.000 deg,	R =   90.000 deg
};
P[178]{
   GP1:
	UF : 0, UT : 6,		CONFIG : 'N U T, 0, 0, 0',
	X =  203.243  mm,	Y =   -321.380  mm,	Z =   -329.100  mm,
	W =  90.000 deg,	P =   0.000 deg,	R =   90.000 deg
};
P[179]{
   GP1:
	UF : 0, UT : 6,		CONFIG : 'N U T, 0, 0, 0',
	X =  204.045  mm,	Y =   -320.686  mm,	Z =   -329.100  mm,
	W =  90.000 deg,	P =   0.000 deg,	R =   90.000 deg
};
P[180]{
   GP1:
	UF : 0, UT : 6,		CONFIG : 'N U T, 0, 0, 0',
	X =  205.473  mm,	Y =   -320.332  mm,	Z =   -329.671  mm,
	W =  90.000 deg,	P =   0.000 deg,	R =   90.000 deg
};
P[181]{
   GP1:
	UF : 0, UT : 6,		CONFIG : 'N U T, 0, 0, 0',
	X =  205.769  mm,	Y =   -319.592  mm,	Z =   -329.100  mm,
	W =  90.000 deg,	P =   0.000 deg,	R =   90.000 deg
};
P[182]{
   GP1:
	UF : 0, UT : 6,		CONFIG : 'N U T, 0, 0, 0',
	X =  206.052  mm,	Y =   -320.071  mm,	Z =   -331.610  mm,
	W =  90.000 deg,	P =   0.000 deg,	R =   90.000 deg
};
P[183]{
   GP1:
	UF : 0, UT : 6,		CONFIG : 'N U T, 0, 0, 0',
	X =  206.043  mm,	Y =   -319.904  mm,	Z =   -330.151  mm,
	W =  90.000 deg,	P =   0.000 deg,	R =   90.000 deg
};
P[184]{
   GP1:
	UF : 0, UT : 6,		CONFIG : 'N U T, 0, 0, 0',
	X =  206.290  mm,	Y =   -319.791  mm,	Z =   -330.936  mm,
	W =  90.000 deg,	P =   0.000 deg,	R =   90.000 deg
};
P[185]{
   GP1:
	UF : 0, UT : 6,		CONFIG : 'N U T, 0, 0, 0',
	X =  206.668  mm,	Y =   -319.359  mm,	Z =   -329.977  mm,
	W =  90.000 deg,	P =   0.000 deg,	R =   90.000 deg
};
P[186]{
   GP1:
	UF : 0, UT : 6,		CONFIG : 'N U T, 0, 0, 0',
	X =  206.862  mm,	Y =   -319.309  mm,	Z =   -330.941  mm,
	W =  90.000 deg,	P =   0.000 deg,	R =   90.000 deg
};
P[187]{
   GP1:
	UF : 0, UT : 6,		CONFIG : 'N U T, 0, 0, 0',
	X =  207.141  mm,	Y =   -319.172  mm,	Z =   -331.684  mm,
	W =  90.000 deg,	P =   0.000 deg,	R =   90.000 deg
};
P[188]{
   GP1:
	UF : 0, UT : 6,		CONFIG : 'N U T, 0, 0, 0',
	X =  207.203  mm,	Y =   -318.782  mm,	Z =   -329.100  mm,
	W =  90.000 deg,	P =   0.000 deg,	R =   90.000 deg
};
P[189]{
   GP1:
	UF : 0, UT : 6,		CONFIG : 'N U T, 0, 0, 0',
	X =  207.303  mm,	Y =   -318.821  mm,	Z =   -329.933  mm,
	W =  90.000 deg,	P =   0.000 deg,	R =   90.000 deg
};
P[190]{
   GP1:
	UF : 0, UT : 6,		CONFIG : 'N U T, 0, 0, 0',
	X =  207.631  mm,	Y =   -318.926  mm,	Z =   -332.257  mm,
	W =  90.000 deg,	P =   0.000 deg,	R =   90.000 deg
};
P[191]{
   GP1:
	UF : 0, UT : 6,		CONFIG : 'N U T, 0, 0, 0',
	X =  207.665  mm,	Y =   -318.643  mm,	Z =   -331.022  mm,
	W =  90.000 deg,	P =   0.000 deg,	R =   90.000 deg
};
P[192]{
   GP1:
	UF : 0, UT : 6,		CONFIG : 'N U T, 0, 0, 0',
	X =  208.032  mm,	Y =   -318.939  mm,	Z =   -333.293  mm,
	W =  90.000 deg,	P =   0.000 deg,	R =   90.000 deg
};
P[193]{
   GP1:
	UF : 0, UT : 6,		CONFIG : 'N U T, 0, 0, 0',
	X =  207.889  mm,	Y =   -318.306  mm,	Z =   -329.683  mm,
	W =  90.000 deg,	P =   0.000 deg,	R =   90.000 deg
};
P[194]{
   GP1:
	UF : 0, UT : 6,		CONFIG : 'N U T, 0, 0, 0',
	X =  208.340  mm,	Y =   -318.080  mm,	Z =   -331.060  mm,
	W =  90.000 deg,	P =   0.000 deg,	R =   90.000 deg
};
P[195]{
   GP1:
	UF : 0, UT : 6,		CONFIG : 'N U T, 0, 0, 0',
	X =  208.460  mm,	Y =   -318.272  mm,	Z =   -332.414  mm,
	W =  90.000 deg,	P =   0.000 deg,	R =   90.000 deg
};
P[196]{
   GP1:
	UF : 0, UT : 6,		CONFIG : 'N U T, 0, 0, 0',
	X =  208.820  mm,	Y =   -318.370  mm,	Z =   -333.571  mm,
	W =  90.000 deg,	P =   0.000 deg,	R =   90.000 deg
};
P[197]{
   GP1:
	UF : 0, UT : 6,		CONFIG : 'N U T, 0, 0, 0',
	X =  208.544  mm,	Y =   -317.735  mm,	Z =   -329.459  mm,
	W =  90.000 deg,	P =   0.000 deg,	R =   90.000 deg
};
P[198]{
   GP1:
	UF : 0, UT : 6,		CONFIG : 'N U T, 0, 0, 0',
	X =  208.984  mm,	Y =   -317.416  mm,	Z =   -329.984  mm,
	W =  90.000 deg,	P =   0.000 deg,	R =   90.000 deg
};
P[199]{
   GP1:
	UF : 0, UT : 6,		CONFIG : 'N U T, 0, 0, 0',
	X =  209.296  mm,	Y =   -317.771  mm,	Z =   -333.049  mm,
	W =  90.000 deg,	P =   0.000 deg,	R =   90.000 deg
};
P[200]{
   GP1:
	UF : 0, UT : 6,		CONFIG : 'N U T, 0, 0, 0',
	X =  209.202  mm,	Y =   -317.597  mm,	Z =   -332.250  mm,
	W =  90.000 deg,	P =   0.000 deg,	R =   90.000 deg
};
P[201]{
   GP1:
	UF : 0, UT : 6,		CONFIG : 'N U T, 0, 0, 0',
	X =  209.213  mm,	Y =   -317.349  mm,	Z =   -331.082  mm,
	W =  90.000 deg,	P =   0.000 deg,	R =   90.000 deg
};
P[202]{
   GP1:
	UF : 0, UT : 6,		CONFIG : 'N U T, 0, 0, 0',
	X =  209.610  mm,	Y =   -317.986  mm,	Z =   -334.311  mm,
	W =  90.000 deg,	P =   0.000 deg,	R =   90.000 deg
};
P[203]{
   GP1:
	UF : 0, UT : 6,		CONFIG : 'N U T, 0, 0, 0',
	X =  210.034  mm,	Y =   -317.482  mm,	Z =   -333.977  mm,
	W =  90.000 deg,	P =   0.000 deg,	R =   90.000 deg
};
P[204]{
   GP1:
	UF : 0, UT : 6,		CONFIG : 'N U T, 0, 0, 0',
	X =  209.721  mm,	Y =   -316.920  mm,	Z =   -331.079  mm,
	W =  90.000 deg,	P =   0.000 deg,	R =   90.000 deg
};
P[205]{
   GP1:
	UF : 0, UT : 6,		CONFIG : 'N U T, 0, 0, 0',
	X =  209.844  mm,	Y =   -317.107  mm,	Z =   -332.425  mm,
	W =  90.000 deg,	P =   0.000 deg,	R =   90.000 deg
};
P[206]{
   GP1:
	UF : 0, UT : 6,		CONFIG : 'N U T, 0, 0, 0',
	X =  210.183  mm,	Y =   -317.131  mm,	Z =   -333.365  mm,
	W =  90.000 deg,	P =   0.000 deg,	R =   90.000 deg
};
P[207]{
   GP1:
	UF : 0, UT : 6,		CONFIG : 'N U T, 0, 0, 0',
	X =  210.905  mm,	Y =   -317.122  mm,	Z =   -334.798  mm,
	W =  90.000 deg,	P =   0.000 deg,	R =   90.000 deg
};
P[208]{
   GP1:
	UF : 0, UT : 6,		CONFIG : 'N U T, 0, 0, 0',
	X =  210.770  mm,	Y =   -316.421  mm,	Z =   -332.755  mm,
	W =  90.000 deg,	P =   0.000 deg,	R =   90.000 deg
};
P[209]{
   GP1:
	UF : 0, UT : 6,		CONFIG : 'N U T, 0, 0, 0',
	X =  211.326  mm,	Y =   -316.334  mm,	Z =   -333.852  mm,
	W =  90.000 deg,	P =   0.000 deg,	R =   90.000 deg
};
P[210]{
   GP1:
	UF : 0, UT : 6,		CONFIG : 'N U T, 0, 0, 0',
	X =  211.986  mm,	Y =   -316.418  mm,	Z =   -335.236  mm,
	W =  90.000 deg,	P =   0.000 deg,	R =   90.000 deg
};
P[211]{
   GP1:
	UF : 0, UT : 6,		CONFIG : 'N U T, 0, 0, 0',
	X =  212.042  mm,	Y =   -315.771  mm,	Z =   -333.981  mm,
	W =  90.000 deg,	P =   0.000 deg,	R =   90.000 deg
};
P[212]{
   GP1:
	UF : 0, UT : 6,		CONFIG : 'N U T, 0, 0, 0',
	X =  213.076  mm,	Y =   -315.923  mm,	Z =   -336.014  mm,
	W =  90.000 deg,	P =   0.000 deg,	R =   90.000 deg
};
P[213]{
   GP1:
	UF : 0, UT : 6,		CONFIG : 'N U T, 0, 0, 0',
	X =  212.878  mm,	Y =   -315.162  mm,	Z =   -334.268  mm,
	W =  90.000 deg,	P =   0.000 deg,	R =   90.000 deg
};
P[214]{
   GP1:
	UF : 0, UT : 6,		CONFIG : 'N U T, 0, 0, 0',
	X =  213.089  mm,	Y =   -315.365  mm,	Z =   -335.029  mm,
	W =  90.000 deg,	P =   0.000 deg,	R =   90.000 deg
};
P[215]{
   GP1:
	UF : 0, UT : 6,		CONFIG : 'N U T, 0, 0, 0',
	X =  213.731  mm,	Y =   -315.379  mm,	Z =   -336.057  mm,
	W =  90.000 deg,	P =   0.000 deg,	R =   90.000 deg
};
P[216]{
   GP1:
	UF : 0, UT : 6,		CONFIG : 'N U T, 0, 0, 0',
	X =  213.744  mm,	Y =   -314.849  mm,	Z =   -335.118  mm,
	W =  90.000 deg,	P =   0.000 deg,	R =   90.000 deg
};
P[217]{
   GP1:
	UF : 0, UT : 6,		CONFIG : 'N U T, 0, 0, 0',
	X =  214.547  mm,	Y =   -314.674  mm,	Z =   -336.058  mm,
	W =  90.000 deg,	P =   0.000 deg,	R =   90.000 deg
};
P[218]{
   GP1:
	UF : 0, UT : 6,		CONFIG : 'N U T, 0, 0, 0',
	X =  214.610  mm,	Y =   -314.055  mm,	Z =   -335.019  mm,
	W =  90.000 deg,	P =   0.000 deg,	R =   90.000 deg
};
P[219]{
   GP1:
	UF : 0, UT : 6,		CONFIG : 'N U T, 0, 0, 0',
	X =  215.470  mm,	Y =   -314.676  mm,	Z =   -337.254  mm,
	W =  90.000 deg,	P =   0.000 deg,	R =   90.000 deg
};
P[220]{
   GP1:
	UF : 0, UT : 6,		CONFIG : 'N U T, 0, 0, 0',
	X =  215.253  mm,	Y =   -314.105  mm,	Z =   -336.117  mm,
	W =  90.000 deg,	P =   0.000 deg,	R =   90.000 deg
};
P[221]{
   GP1:
	UF : 0, UT : 6,		CONFIG : 'N U T, 0, 0, 0',
	X =  215.942  mm,	Y =   -313.523  mm,	Z =   -336.173  mm,
	W =  90.000 deg,	P =   0.000 deg,	R =   90.000 deg
};
P[222]{
   GP1:
	UF : 0, UT : 6,		CONFIG : 'N U T, 0, 0, 0',
	X =  216.430  mm,	Y =   -313.527  mm,	Z =   -336.853  mm,
	W =  90.000 deg,	P =   0.000 deg,	R =   90.000 deg
};
P[223]{
   GP1:
	UF : 0, UT : 6,		CONFIG : 'N U T, 0, 0, 0',
	X =  216.936  mm,	Y =   -313.722  mm,	Z =   -337.704  mm,
	W =  90.000 deg,	P =   0.000 deg,	R =   90.000 deg
};
P[224]{
   GP1:
	UF : 0, UT : 6,		CONFIG : 'N U T, 0, 0, 0',
	X =  217.030  mm,	Y =   -313.216  mm,	Z =   -337.145  mm,
	W =  90.000 deg,	P =   0.000 deg,	R =   90.000 deg
};
P[225]{
   GP1:
	UF : 0, UT : 6,		CONFIG : 'N U T, 0, 0, 0',
	X =  218.023  mm,	Y =   -313.163  mm,	Z =   -338.235  mm,
	W =  90.000 deg,	P =   0.000 deg,	R =   90.000 deg
};
P[226]{
   GP1:
	UF : 0, UT : 6,		CONFIG : 'N U T, 0, 0, 0',
	X =  217.773  mm,	Y =   -312.558  mm,	Z =   -337.140  mm,
	W =  90.000 deg,	P =   0.000 deg,	R =   90.000 deg
};
P[227]{
   GP1:
	UF : 0, UT : 6,		CONFIG : 'N U T, 0, 0, 0',
	X =  218.845  mm,	Y =   -312.189  mm,	Z =   -337.905  mm,
	W =  90.000 deg,	P =   0.000 deg,	R =   90.000 deg
};
P[228]{
   GP1:
	UF : 0, UT : 6,		CONFIG : 'N U T, 0, 0, 0',
	X =  218.775  mm,	Y =   -311.690  mm,	Z =   -337.163  mm,
	W =  90.000 deg,	P =   0.000 deg,	R =   90.000 deg
};
P[229]{
   GP1:
	UF : 0, UT : 6,		CONFIG : 'N U T, 0, 0, 0',
	X =  219.492  mm,	Y =   -311.576  mm,	Z =   -337.849  mm,
	W =  90.000 deg,	P =   0.000 deg,	R =   90.000 deg
};
P[230]{
   GP1:
	UF : 0, UT : 6,		CONFIG : 'N U T, 0, 0, 0',
	X =  219.810  mm,	Y =   -311.980  mm,	Z =   -338.755  mm,
	W =  90.000 deg,	P =   0.000 deg,	R =   90.000 deg
};
P[231]{
   GP1:
	UF : 0, UT : 6,		CONFIG : 'N U T, 0, 0, 0',
	X =  220.337  mm,	Y =   -310.904  mm,	Z =   -337.947  mm,
	W =  90.000 deg,	P =   0.000 deg,	R =   90.000 deg
};
P[232]{
   GP1:
	UF : 0, UT : 6,		CONFIG : 'N U T, 0, 0, 0',
	X =  220.764  mm,	Y =   -311.522  mm,	Z =   -339.204  mm,
	W =  90.000 deg,	P =   0.000 deg,	R =   90.000 deg
};
P[233]{
   GP1:
	UF : 0, UT : 6,		CONFIG : 'N U T, 0, 0, 0',
	X =  221.323  mm,	Y =   -310.905  mm,	Z =   -339.058  mm,
	W =  90.000 deg,	P =   0.000 deg,	R =   90.000 deg
};
P[234]{
   GP1:
	UF : 0, UT : 6,		CONFIG : 'N U T, 0, 0, 0',
	X =  221.591  mm,	Y =   -310.193  mm,	Z =   -338.470  mm,
	W =  90.000 deg,	P =   0.000 deg,	R =   90.000 deg
};
P[235]{
   GP1:
	UF : 0, UT : 6,		CONFIG : 'N U T, 0, 0, 0',
	X =  222.470  mm,	Y =   -310.395  mm,	Z =   -339.635  mm,
	W =  90.000 deg,	P =   0.000 deg,	R =   90.000 deg
};
P[236]{
   GP1:
	UF : 0, UT : 6,		CONFIG : 'N U T, 0, 0, 0',
	X =  222.386  mm,	Y =   -309.858  mm,	Z =   -338.958  mm,
	W =  90.000 deg,	P =   0.000 deg,	R =   90.000 deg
};
P[237]{
   GP1:
	UF : 0, UT : 6,		CONFIG : 'N U T, 0, 0, 0',
	X =  222.946  mm,	Y =   -309.827  mm,	Z =   -339.510  mm,
	W =  90.000 deg,	P =   0.000 deg,	R =   90.000 deg
};
P[238]{
   GP1:
	UF : 0, UT : 6,		CONFIG : 'N U T, 0, 0, 0',
	X =  223.360  mm,	Y =   -309.141  mm,	Z =   -339.146  mm,
	W =  90.000 deg,	P =   0.000 deg,	R =   90.000 deg
};
P[239]{
   GP1:
	UF : 0, UT : 6,		CONFIG : 'N U T, 0, 0, 0',
	X =  223.980  mm,	Y =   -309.427  mm,	Z =   -340.036  mm,
	W =  90.000 deg,	P =   0.000 deg,	R =   90.000 deg
};
P[240]{
   GP1:
	UF : 0, UT : 6,		CONFIG : 'N U T, 0, 0, 0',
	X =  224.639  mm,	Y =   -308.294  mm,	Z =   -339.517  mm,
	W =  90.000 deg,	P =   0.000 deg,	R =   90.000 deg
};
P[241]{
   GP1:
	UF : 0, UT : 6,		CONFIG : 'N U T, 0, 0, 0',
	X =  225.168  mm,	Y =   -308.692  mm,	Z =   -340.375  mm,
	W =  90.000 deg,	P =   0.000 deg,	R =   90.000 deg
};
P[242]{
   GP1:
	UF : 0, UT : 6,		CONFIG : 'N U T, 0, 0, 0',
	X =  225.703  mm,	Y =   -308.761  mm,	Z =   -340.906  mm,
	W =  90.000 deg,	P =   0.000 deg,	R =   90.000 deg
};
P[243]{
   GP1:
	UF : 0, UT : 6,		CONFIG : 'N U T, 0, 0, 0',
	X =  225.619  mm,	Y =   -307.843  mm,	Z =   -339.966  mm,
	W =  90.000 deg,	P =   0.000 deg,	R =   90.000 deg
};
P[244]{
   GP1:
	UF : 0, UT : 6,		CONFIG : 'N U T, 0, 0, 0',
	X =  226.601  mm,	Y =   -307.845  mm,	Z =   -340.822  mm,
	W =  90.000 deg,	P =   0.000 deg,	R =   90.000 deg
};
P[245]{
   GP1:
	UF : 0, UT : 6,		CONFIG : 'N U T, 0, 0, 0',
	X =  226.874  mm,	Y =   -306.997  mm,	Z =   -340.161  mm,
	W =  90.000 deg,	P =   0.000 deg,	R =   90.000 deg
};
P[246]{
   GP1:
	UF : 0, UT : 6,		CONFIG : 'N U T, 0, 0, 0',
	X =  227.657  mm,	Y =   -307.026  mm,	Z =   -340.612  mm,
	W =  90.000 deg,	P =   0.000 deg,	R =   90.000 deg
};
P[247]{
   GP1:
	UF : 0, UT : 6,		CONFIG : 'N U T, 0, 0, 0',
	X =  228.494  mm,	Y =   -306.802  mm,	Z =   -340.804  mm,
	W =  90.000 deg,	P =   0.000 deg,	R =   90.000 deg
};
P[248]{
   GP1:
	UF : 0, UT : 6,		CONFIG : 'N U T, 0, 0, 0',
	X =  229.458  mm,	Y =   -306.403  mm,	Z =   -340.865  mm,
	W =  90.000 deg,	P =   0.000 deg,	R =   90.000 deg
};
P[249]{
   GP1:
	UF : 0, UT : 6,		CONFIG : 'N U T, 0, 0, 0',
	X =  229.950  mm,	Y =   -305.638  mm,	Z =   -340.255  mm,
	W =  90.000 deg,	P =   0.000 deg,	R =   90.000 deg
};
P[250]{
   GP1:
	UF : 0, UT : 6,		CONFIG : 'N U T, 0, 0, 0',
	X =  230.891  mm,	Y =   -305.103  mm,	Z =   -340.072  mm,
	W =  90.000 deg,	P =   0.000 deg,	R =   90.000 deg
};
P[251]{
   GP1:
	UF : 0, UT : 6,		CONFIG : 'N U T, 0, 0, 0',
	X =  231.184  mm,	Y =   -304.565  mm,	Z =   -339.519  mm,
	W =  90.000 deg,	P =   0.000 deg,	R =   90.000 deg
};
P[252]{
   GP1:
	UF : 0, UT : 6,		CONFIG : 'N U T, 0, 0, 0',
	X =  232.000  mm,	Y =   -305.016  mm,	Z =   -340.411  mm,
	W =  90.000 deg,	P =   0.000 deg,	R =   90.000 deg
};
P[253]{
   GP1:
	UF : 0, UT : 6,		CONFIG : 'N U T, 0, 0, 0',
	X =  232.548  mm,	Y =   -304.482  mm,	Z =   -339.981  mm,
	W =  90.000 deg,	P =   0.000 deg,	R =   90.000 deg
};
P[254]{
   GP1:
	UF : 0, UT : 6,		CONFIG : 'N U T, 0, 0, 0',
	X =  232.987  mm,	Y =   -303.914  mm,	Z =   -339.465  mm,
	W =  90.000 deg,	P =   0.000 deg,	R =   90.000 deg
};
P[255]{
   GP1:
	UF : 0, UT : 6,		CONFIG : 'N U T, 0, 0, 0',
	X =  233.485  mm,	Y =   -303.456  mm,	Z =   -339.018  mm,
	W =  90.000 deg,	P =   0.000 deg,	R =   90.000 deg
};
P[256]{
   GP1:
	UF : 0, UT : 6,		CONFIG : 'N U T, 0, 0, 0',
	X =  233.783  mm,	Y =   -303.961  mm,	Z =   -339.843  mm,
	W =  90.000 deg,	P =   0.000 deg,	R =   90.000 deg
};
P[257]{
   GP1:
	UF : 0, UT : 6,		CONFIG : 'N U T, 0, 0, 0',
	X =  234.767  mm,	Y =   -303.183  mm,	Z =   -339.118  mm,
	W =  90.000 deg,	P =   0.000 deg,	R =   90.000 deg
};
P[258]{
   GP1:
	UF : 0, UT : 6,		CONFIG : 'N U T, 0, 0, 0',
	X =  235.463  mm,	Y =   -302.904  mm,	Z =   -338.950  mm,
	W =  90.000 deg,	P =   0.000 deg,	R =   90.000 deg
};
P[259]{
   GP1:
	UF : 0, UT : 6,		CONFIG : 'N U T, 0, 0, 0',
	X =  235.566  mm,	Y =   -302.295  mm,	Z =   -337.943  mm,
	W =  90.000 deg,	P =   0.000 deg,	R =   90.000 deg
};
P[260]{
   GP1:
	UF : 0, UT : 6,		CONFIG : 'N U T, 0, 0, 0',
	X =  236.417  mm,	Y =   -302.288  mm,	Z =   -338.284  mm,
	W =  90.000 deg,	P =   0.000 deg,	R =   90.000 deg
};
P[261]{
   GP1:
	UF : 0, UT : 6,		CONFIG : 'N U T, 0, 0, 0',
	X =  236.228  mm,	Y =   -301.886  mm,	Z =   -337.497  mm,
	W =  90.000 deg,	P =   0.000 deg,	R =   90.000 deg
};
P[262]{
   GP1:
	UF : 0, UT : 6,		CONFIG : 'N U T, 0, 0, 0',
	X =  237.295  mm,	Y =   -301.473  mm,	Z =   -337.209  mm,
	W =  90.000 deg,	P =   0.000 deg,	R =   90.000 deg
};
P[263]{
   GP1:
	UF : 0, UT : 6,		CONFIG : 'N U T, 0, 0, 0',
	X =  237.654  mm,	Y =   -300.931  mm,	Z =   -336.269  mm,
	W =  90.000 deg,	P =   0.000 deg,	R =   90.000 deg
};
P[264]{
   GP1:
	UF : 0, UT : 6,		CONFIG : 'N U T, 0, 0, 0',
	X =  238.148  mm,	Y =   -301.096  mm,	Z =   -336.775  mm,
	W =  90.000 deg,	P =   0.000 deg,	R =   90.000 deg
};
P[265]{
   GP1:
	UF : 0, UT : 6,		CONFIG : 'N U T, 0, 0, 0',
	X =  238.861  mm,	Y =   -300.634  mm,	Z =   -335.993  mm,
	W =  90.000 deg,	P =   0.000 deg,	R =   90.000 deg
};
P[266]{
   GP1:
	UF : 0, UT : 6,		CONFIG : 'N U T, 0, 0, 0',
	X =  238.775  mm,	Y =   -300.357  mm,	Z =   -335.208  mm,
	W =  90.000 deg,	P =   0.000 deg,	R =   90.000 deg
};
P[267]{
   GP1:
	UF : 0, UT : 6,		CONFIG : 'N U T, 0, 0, 0',
	X =  238.734  mm,	Y =   -300.111  mm,	Z =   -334.524  mm,
	W =  90.000 deg,	P =   0.000 deg,	R =   90.000 deg
};
P[268]{
   GP1:
	UF : 0, UT : 6,		CONFIG : 'N U T, 0, 0, 0',
	X =  239.476  mm,	Y =   -299.854  mm,	Z =   -334.116  mm,
	W =  90.000 deg,	P =   0.000 deg,	R =   90.000 deg
};
P[269]{
   GP1:
	UF : 0, UT : 6,		CONFIG : 'N U T, 0, 0, 0',
	X =  239.942  mm,	Y =   -300.263  mm,	Z =   -335.430  mm,
	W =  90.000 deg,	P =   0.000 deg,	R =   90.000 deg
};
P[270]{
   GP1:
	UF : 0, UT : 6,		CONFIG : 'N U T, 0, 0, 0',
	X =  240.061  mm,	Y =   -299.686  mm,	Z =   -333.917  mm,
	W =  90.000 deg,	P =   0.000 deg,	R =   90.000 deg
};
P[271]{
   GP1:
	UF : 0, UT : 6,		CONFIG : 'N U T, 0, 0, 0',
	X =  240.485  mm,	Y =   -300.018  mm,	Z =   -334.986  mm,
	W =  90.000 deg,	P =   0.000 deg,	R =   90.000 deg
};
P[272]{
   GP1:
	UF : 0, UT : 6,		CONFIG : 'N U T, 0, 0, 0',
	X =  240.290  mm,	Y =   -299.505  mm,	Z =   -333.335  mm,
	W =  90.000 deg,	P =   0.000 deg,	R =   90.000 deg
};
P[273]{
   GP1:
	UF : 0, UT : 6,		CONFIG : 'N U T, 0, 0, 0',
	X =  240.305  mm,	Y =   -299.223  mm,	Z =   -332.048  mm,
	W =  90.000 deg,	P =   0.000 deg,	R =   90.000 deg
};
P[274]{
   GP1:
	UF : 0, UT : 6,		CONFIG : 'N U T, 0, 0, 0',
	X =  241.051  mm,	Y =   -298.947  mm,	Z =   -330.844  mm,
	W =  90.000 deg,	P =   0.000 deg,	R =   90.000 deg
};
P[275]{
   GP1:
	UF : 0, UT : 6,		CONFIG : 'N U T, 0, 0, 0',
	X =  241.399  mm,	Y =   -299.549  mm,	Z =   -334.014  mm,
	W =  90.000 deg,	P =   0.000 deg,	R =   90.000 deg
};
P[276]{
   GP1:
	UF : 0, UT : 6,		CONFIG : 'N U T, 0, 0, 0',
	X =  241.150  mm,	Y =   -299.115  mm,	Z =   -332.074  mm,
	W =  90.000 deg,	P =   0.000 deg,	R =   90.000 deg
};
P[277]{
   GP1:
	UF : 0, UT : 6,		CONFIG : 'N U T, 0, 0, 0',
	X =  241.428  mm,	Y =   -298.837  mm,	Z =   -329.654  mm,
	W =  90.000 deg,	P =   0.000 deg,	R =   90.000 deg
};
P[278]{
   GP1:
	UF : 0, UT : 6,		CONFIG : 'N U T, 0, 0, 0',
	X =  242.083  mm,	Y =   -299.067  mm,	Z =   -332.152  mm,
	W =  90.000 deg,	P =   0.000 deg,	R =   90.000 deg
};
P[279]{
   GP1:
	UF : 0, UT : 6,		CONFIG : 'N U T, 0, 0, 0',
	X =  242.167  mm,	Y =   -298.868  mm,	Z =   -330.957  mm,
	W =  90.000 deg,	P =   0.000 deg,	R =   90.000 deg
};
P[280]{
   GP1:
	UF : 0, UT : 6,		CONFIG : 'N U T, 0, 0, 0',
	X =  242.205  mm,	Y =   -298.592  mm,	Z =   -329.100  mm,
	W =  90.000 deg,	P =   0.000 deg,	R =   90.000 deg
};
P[281]{
   GP1:
	UF : 0, UT : 6,		CONFIG : 'N U T, 0, 0, 0',
	X =  242.597  mm,	Y =   -298.782  mm,	Z =   -330.174  mm,
	W =  90.000 deg,	P =   0.000 deg,	R =   90.000 deg
};
P[282]{
   GP1:
	UF : 0, UT : 6,		CONFIG : 'N U T, 0, 0, 0',
	X =  242.944  mm,	Y =   -298.332  mm,	Z =   -329.100  mm,
	W =  90.000 deg,	P =   0.000 deg,	R =   90.000 deg
};
P[283]{
   GP1:
	UF : 0, UT : 6,		CONFIG : 'N U T, 0, 0, 0',
	X =  243.482  mm,	Y =   -297.676  mm,	Z =   -329.100  mm,
	W =  90.000 deg,	P =   0.000 deg,	R =   90.000 deg
};
P[284]{
   GP1:
	UF : 0, UT : 6,		CONFIG : 'N U T, 0, 0, 0',
	X =  244.682  mm,	Y =   -297.198  mm,	Z =   -329.100  mm,
	W =  90.000 deg,	P =   0.000 deg,	R =   90.000 deg
};
P[285]{
   GP1:
	UF : 0, UT : 6,		CONFIG : 'N U T, 0, 0, 0',
	X =  245.574  mm,	Y =   -296.432  mm,	Z =   -329.100  mm,
	W =  90.000 deg,	P =   0.000 deg,	R =   90.000 deg
};
P[286]{
   GP1:
	UF : 0, UT : 6,		CONFIG : 'N U T, 0, 0, 0',
	X =  246.940  mm,	Y =   -296.327  mm,	Z =   -329.100  mm,
	W =  90.000 deg,	P =   0.000 deg,	R =   90.000 deg
};
P[287]{
   GP1:
	UF : 0, UT : 6,		CONFIG : 'N U T, 0, 0, 0',
	X =  247.428  mm,	Y =   -295.723  mm,	Z =   -329.100  mm,
	W =  90.000 deg,	P =   0.000 deg,	R =   90.000 deg
};
P[288]{
   GP1:
	UF : 0, UT : 6,		CONFIG : 'N U T, 0, 0, 0',
	X =  249.150  mm,	Y =   -294.954  mm,	Z =   -329.100  mm,
	W =  90.000 deg,	P =   0.000 deg,	R =   90.000 deg
};
P[289]{
   GP1:
	UF : 0, UT : 6,		CONFIG : 'N U T, 0, 0, 0',
	X =  250.537  mm,	Y =   -294.080  mm,	Z =   -329.100  mm,
	W =  90.000 deg,	P =   0.000 deg,	R =   90.000 deg
};
P[290]{
   GP1:
	UF : 0, UT : 6,		CONFIG : 'N U T, 0, 0, 0',
	X =  252.499  mm,	Y =   -292.892  mm,	Z =   -329.100  mm,
	W =  90.000 deg,	P =   0.000 deg,	R =   90.000 deg
};
P[291]{
   GP1:
	UF : 0, UT : 6,		CONFIG : 'N U T, 0, 0, 0',
	X =  253.274  mm,	Y =   -292.236  mm,	Z =   -329.100  mm,
	W =  90.000 deg,	P =   0.000 deg,	R =   90.000 deg
};
P[292]{
   GP1:
	UF : 0, UT : 6,		CONFIG : 'N U T, 0, 0, 0',
	X =  254.048  mm,	Y =   -291.782  mm,	Z =   -329.100  mm,
	W =  90.000 deg,	P =   0.000 deg,	R =   90.000 deg
};
P[293]{
   GP1:
	UF : 0, UT : 6,		CONFIG : 'N U T, 0, 0, 0',
	X =  255.095  mm,	Y =   -291.250  mm,	Z =   -329.100  mm,
	W =  90.000 deg,	P =   0.000 deg,	R =   90.000 deg
};
P[294]{
   GP1:
	UF : 0, UT : 6,		CONFIG : 'N U T, 0, 0, 0',
	X =  255.921  mm,	Y =   -290.548  mm,	Z =   -329.100  mm,
	W =  90.000 deg,	P =   0.000 deg,	R =   90.000 deg
};
P[295]{
   GP1:
	UF : 0, UT : 6,		CONFIG : 'N U T, 0, 0, 0',
	X =  257.027  mm,	Y =   -290.217  mm,	Z =   -329.100  mm,
	W =  90.000 deg,	P =   0.000 deg,	R =   90.000 deg
};
P[296]{
   GP1:
	UF : 0, UT : 6,		CONFIG : 'N U T, 0, 0, 0',
	X =  258.885  mm,	Y =   -289.445  mm,	Z =   -329.000  mm,
	W =  90.000 deg,	P =   0.000 deg,	R =   90.000 deg
};
P[297]{
   GP1:
	UF : 0, UT : 6,		CONFIG : 'N U T, 0, 0, 0',
	X =  259.490  mm,	Y =   -288.981  mm,	Z =   -329.000  mm,
	W =  90.000 deg,	P =   0.000 deg,	R =   90.000 deg
};
P[298]{
   GP1:
	UF : 0, UT : 6,		CONFIG : 'N U T, 0, 0, 0',
	X =  260.132  mm,	Y =   -288.239  mm,	Z =   -329.000  mm,
	W =  90.000 deg,	P =   0.000 deg,	R =   90.000 deg
};
P[299]{
   GP1:
	UF : 0, UT : 6,		CONFIG : 'N U T, 0, 0, 0',
	X =  261.345  mm,	Y =   -287.914  mm,	Z =   -329.000  mm,
	W =  90.000 deg,	P =   0.000 deg,	R =   90.000 deg
};
P[300]{
   GP1:
	UF : 0, UT : 6,		CONFIG : 'N U T, 0, 0, 0',
	X =  261.957  mm,	Y =   -286.871  mm,	Z =   -329.000  mm,
	W =  90.000 deg,	P =   0.000 deg,	R =   90.000 deg
};
P[301]{
   GP1:
	UF : 0, UT : 6,		CONFIG : 'N U T, 0, 0, 0',
	X =  263.681  mm,	Y =   -286.004  mm,	Z =   -329.000  mm,
	W =  90.000 deg,	P =   0.000 deg,	R =   90.000 deg
};
P[302]{
   GP1:
	UF : 0, UT : 6,		CONFIG : 'N U T, 0, 0, 0',
	X =  264.943  mm,	Y =   -285.590  mm,	Z =   -329.000  mm,
	W =  90.000 deg,	P =   0.000 deg,	R =   90.000 deg
};
P[303]{
   GP1:
	UF : 0, UT : 6,		CONFIG : 'N U T, 0, 0, 0',
	X =  266.140  mm,	Y =   -284.795  mm,	Z =   -329.000  mm,
	W =  90.000 deg,	P =   0.000 deg,	R =   90.000 deg
};
P[304]{
   GP1:
	UF : 0, UT : 6,		CONFIG : 'N U T, 0, 0, 0',
	X =  267.083  mm,	Y =   -284.746  mm,	Z =   -329.000  mm,
	W =  90.000 deg,	P =   0.000 deg,	R =   90.000 deg
};
P[305]{
   GP1:
	UF : 0, UT : 6,		CONFIG : 'N U T, 0, 0, 0',
	X =  268.276  mm,	Y =   -283.615  mm,	Z =   -329.000  mm,
	W =  90.000 deg,	P =   0.000 deg,	R =   90.000 deg
};
P[306]{
   GP1:
	UF : 0, UT : 6,		CONFIG : 'N U T, 0, 0, 0',
	X =  268.996  mm,	Y =   -282.704  mm,	Z =   -329.000  mm,
	W =  90.000 deg,	P =   0.000 deg,	R =   90.000 deg
};
P[307]{
   GP1:
	UF : 0, UT : 6,		CONFIG : 'N U T, 0, 0, 0',
	X =  269.826  mm,	Y =   -282.937  mm,	Z =   -329.000  mm,
	W =  90.000 deg,	P =   0.000 deg,	R =   90.000 deg
};
P[308]{
   GP1:
	UF : 0, UT : 6,		CONFIG : 'N U T, 0, 0, 0',
	X =  270.851  mm,	Y =   -282.249  mm,	Z =   -329.000  mm,
	W =  90.000 deg,	P =   0.000 deg,	R =   90.000 deg
};
P[309]{
   GP1:
	UF : 0, UT : 6,		CONFIG : 'N U T, 0, 0, 0',
	X =  169.254  mm,	Y =   -341.371  mm,	Z =   -329.100  mm,
	W =  90.000 deg,	P =   0.000 deg,	R =   90.000 deg
};
P[310]{
   GP1:
	UF : 0, UT : 6,		CONFIG : 'N U T, 0, 0, 0',
	X =  149.187  mm,	Y =   -467.668  mm,	Z =   -329.000  mm,
	W =  90.000 deg,	P =   0.000 deg,	R =   90.000 deg
};
P[311]{
   GP1:
	UF : 0, UT : 6,		CONFIG : 'N U T, 0, 0, 0',
	X =  150.449  mm,	Y =   -467.091  mm,	Z =   -329.000  mm,
	W =  90.000 deg,	P =   0.000 deg,	R =   90.000 deg
};
P[312]{
   GP1:
	UF : 0, UT : 6,		CONFIG : 'N U T, 0, 0, 0',
	X =  151.177  mm,	Y =   -467.053  mm,	Z =   -329.000  mm,
	W =  90.000 deg,	P =   0.000 deg,	R =   90.000 deg
};
P[313]{
   GP1:
	UF : 0, UT : 6,		CONFIG : 'N U T, 0, 0, 0',
	X =  152.509  mm,	Y =   -466.040  mm,	Z =   -329.000  mm,
	W =  90.000 deg,	P =   0.000 deg,	R =   90.000 deg
};
P[314]{
   GP1:
	UF : 0, UT : 6,		CONFIG : 'N U T, 0, 0, 0',
	X =  153.161  mm,	Y =   -465.275  mm,	Z =   -329.000  mm,
	W =  90.000 deg,	P =   0.000 deg,	R =   90.000 deg
};
P[315]{
   GP1:
	UF : 0, UT : 6,		CONFIG : 'N U T, 0, 0, 0',
	X =  154.383  mm,	Y =   -464.924  mm,	Z =   -329.000  mm,
	W =  90.000 deg,	P =   0.000 deg,	R =   90.000 deg
};
P[316]{
   GP1:
	UF : 0, UT : 6,		CONFIG : 'N U T, 0, 0, 0',
	X =  155.321  mm,	Y =   -464.363  mm,	Z =   -329.100  mm,
	W =  90.000 deg,	P =   0.000 deg,	R =   90.000 deg
};
P[317]{
   GP1:
	UF : 0, UT : 6,		CONFIG : 'N U T, 0, 0, 0',
	X =  156.016  mm,	Y =   -463.525  mm,	Z =   -329.100  mm,
	W =  90.000 deg,	P =   0.000 deg,	R =   90.000 deg
};
P[318]{
   GP1:
	UF : 0, UT : 6,		CONFIG : 'N U T, 0, 0, 0',
	X =  157.332  mm,	Y =   -463.055  mm,	Z =   -329.100  mm,
	W =  90.000 deg,	P =   0.000 deg,	R =   90.000 deg
};
P[319]{
   GP1:
	UF : 0, UT : 6,		CONFIG : 'N U T, 0, 0, 0',
	X =  158.058  mm,	Y =   -462.429  mm,	Z =   -329.100  mm,
	W =  90.000 deg,	P =   0.000 deg,	R =   90.000 deg
};
P[320]{
   GP1:
	UF : 0, UT : 6,		CONFIG : 'N U T, 0, 0, 0',
	X =  159.187  mm,	Y =   -462.272  mm,	Z =   -329.100  mm,
	W =  90.000 deg,	P =   0.000 deg,	R =   90.000 deg
};
P[321]{
   GP1:
	UF : 0, UT : 6,		CONFIG : 'N U T, 0, 0, 0',
	X =  159.778  mm,	Y =   -461.830  mm,	Z =   -329.100  mm,
	W =  90.000 deg,	P =   0.000 deg,	R =   90.000 deg
};
P[322]{
   GP1:
	UF : 0, UT : 6,		CONFIG : 'N U T, 0, 0, 0',
	X =  160.327  mm,	Y =   -461.159  mm,	Z =   -329.100  mm,
	W =  90.000 deg,	P =   0.000 deg,	R =   90.000 deg
};
P[323]{
   GP1:
	UF : 0, UT : 6,		CONFIG : 'N U T, 0, 0, 0',
	X =  161.330  mm,	Y =   -460.336  mm,	Z =   -329.100  mm,
	W =  90.000 deg,	P =   0.000 deg,	R =   90.000 deg
};
P[324]{
   GP1:
	UF : 0, UT : 6,		CONFIG : 'N U T, 0, 0, 0',
	X =  162.404  mm,	Y =   -460.070  mm,	Z =   -329.100  mm,
	W =  90.000 deg,	P =   0.000 deg,	R =   90.000 deg
};
P[325]{
   GP1:
	UF : 0, UT : 6,		CONFIG : 'N U T, 0, 0, 0',
	X =  163.468  mm,	Y =   -459.770  mm,	Z =   -329.100  mm,
	W =  90.000 deg,	P =   0.000 deg,	R =   90.000 deg
};
P[326]{
   GP1:
	UF : 0, UT : 6,		CONFIG : 'N U T, 0, 0, 0',
	X =  163.783  mm,	Y =   -459.151  mm,	Z =   -329.100  mm,
	W =  90.000 deg,	P =   0.000 deg,	R =   90.000 deg
};
P[327]{
   GP1:
	UF : 0, UT : 6,		CONFIG : 'N U T, 0, 0, 0',
	X =  165.243  mm,	Y =   -458.753  mm,	Z =   -329.100  mm,
	W =  90.000 deg,	P =   0.000 deg,	R =   90.000 deg
};
P[328]{
   GP1:
	UF : 0, UT : 6,		CONFIG : 'N U T, 0, 0, 0',
	X =  165.862  mm,	Y =   -457.656  mm,	Z =   -329.100  mm,
	W =  90.000 deg,	P =   0.000 deg,	R =   90.000 deg
};
P[329]{
   GP1:
	UF : 0, UT : 6,		CONFIG : 'N U T, 0, 0, 0',
	X =  167.331  mm,	Y =   -457.110  mm,	Z =   -329.100  mm,
	W =  90.000 deg,	P =   0.000 deg,	R =   90.000 deg
};
P[330]{
   GP1:
	UF : 0, UT : 6,		CONFIG : 'N U T, 0, 0, 0',
	X =  169.202  mm,	Y =   -456.580  mm,	Z =   -329.100  mm,
	W =  90.000 deg,	P =   0.000 deg,	R =   90.000 deg
};
P[331]{
   GP1:
	UF : 0, UT : 6,		CONFIG : 'N U T, 0, 0, 0',
	X =  169.907  mm,	Y =   -455.702  mm,	Z =   -329.100  mm,
	W =  90.000 deg,	P =   0.000 deg,	R =   90.000 deg
};
P[332]{
   GP1:
	UF : 0, UT : 6,		CONFIG : 'N U T, 0, 0, 0',
	X =  170.948  mm,	Y =   -455.151  mm,	Z =   -329.100  mm,
	W =  90.000 deg,	P =   0.000 deg,	R =   90.000 deg
};
P[333]{
   GP1:
	UF : 0, UT : 6,		CONFIG : 'N U T, 0, 0, 0',
	X =  171.966  mm,	Y =   -454.594  mm,	Z =   -329.100  mm,
	W =  90.000 deg,	P =   0.000 deg,	R =   90.000 deg
};
P[334]{
   GP1:
	UF : 0, UT : 6,		CONFIG : 'N U T, 0, 0, 0',
	X =  172.579  mm,	Y =   -454.034  mm,	Z =   -329.100  mm,
	W =  90.000 deg,	P =   0.000 deg,	R =   90.000 deg
};
P[335]{
   GP1:
	UF : 0, UT : 6,		CONFIG : 'N U T, 0, 0, 0',
	X =  173.398  mm,	Y =   -454.101  mm,	Z =   -329.100  mm,
	W =  90.000 deg,	P =   0.000 deg,	R =   90.000 deg
};
P[336]{
   GP1:
	UF : 0, UT : 6,		CONFIG : 'N U T, 0, 0, 0',
	X =  173.226  mm,	Y =   -453.446  mm,	Z =   -331.334  mm,
	W =  90.000 deg,	P =   0.000 deg,	R =   90.000 deg
};
P[337]{
   GP1:
	UF : 0, UT : 6,		CONFIG : 'N U T, 0, 0, 0',
	X =  173.367  mm,	Y =   -453.524  mm,	Z =   -329.979  mm,
	W =  90.000 deg,	P =   0.000 deg,	R =   90.000 deg
};
P[338]{
   GP1:
	UF : 0, UT : 6,		CONFIG : 'N U T, 0, 0, 0',
	X =  174.098  mm,	Y =   -453.206  mm,	Z =   -330.554  mm,
	W =  90.000 deg,	P =   0.000 deg,	R =   90.000 deg
};
P[339]{
   GP1:
	UF : 0, UT : 6,		CONFIG : 'N U T, 0, 0, 0',
	X =  174.274  mm,	Y =   -453.501  mm,	Z =   -329.320  mm,
	W =  90.000 deg,	P =   0.000 deg,	R =   90.000 deg
};
P[340]{
   GP1:
	UF : 0, UT : 6,		CONFIG : 'N U T, 0, 0, 0',
	X =  174.058  mm,	Y =   -452.992  mm,	Z =   -332.144  mm,
	W =  90.000 deg,	P =   0.000 deg,	R =   90.000 deg
};
P[341]{
   GP1:
	UF : 0, UT : 6,		CONFIG : 'N U T, 0, 0, 0',
	X =  174.506  mm,	Y =   -453.002  mm,	Z =   -331.134  mm,
	W =  90.000 deg,	P =   0.000 deg,	R =   90.000 deg
};
P[342]{
   GP1:
	UF : 0, UT : 6,		CONFIG : 'N U T, 0, 0, 0',
	X =  174.952  mm,	Y =   -452.908  mm,	Z =   -330.437  mm,
	W =  90.000 deg,	P =   0.000 deg,	R =   90.000 deg
};
P[343]{
   GP1:
	UF : 0, UT : 6,		CONFIG : 'N U T, 0, 0, 0',
	X =  174.932  mm,	Y =   -452.753  mm,	Z =   -331.831  mm,
	W =  90.000 deg,	P =   0.000 deg,	R =   90.000 deg
};
P[344]{
   GP1:
	UF : 0, UT : 6,		CONFIG : 'N U T, 0, 0, 0',
	X =  174.955  mm,	Y =   -452.547  mm,	Z =   -332.649  mm,
	W =  90.000 deg,	P =   0.000 deg,	R =   90.000 deg
};
P[345]{
   GP1:
	UF : 0, UT : 6,		CONFIG : 'N U T, 0, 0, 0',
	X =  175.529  mm,	Y =   -453.144  mm,	Z =   -329.100  mm,
	W =  90.000 deg,	P =   0.000 deg,	R =   90.000 deg
};
P[346]{
   GP1:
	UF : 0, UT : 6,		CONFIG : 'N U T, 0, 0, 0',
	X =  175.842  mm,	Y =   -452.560  mm,	Z =   -330.700  mm,
	W =  90.000 deg,	P =   0.000 deg,	R =   90.000 deg
};
P[347]{
   GP1:
	UF : 0, UT : 6,		CONFIG : 'N U T, 0, 0, 0',
	X =  175.647  mm,	Y =   -452.151  mm,	Z =   -333.156  mm,
	W =  90.000 deg,	P =   0.000 deg,	R =   90.000 deg
};
P[348]{
   GP1:
	UF : 0, UT : 6,		CONFIG : 'N U T, 0, 0, 0',
	X =  176.139  mm,	Y =   -452.541  mm,	Z =   -329.700  mm,
	W =  90.000 deg,	P =   0.000 deg,	R =   90.000 deg
};
P[349]{
   GP1:
	UF : 0, UT : 6,		CONFIG : 'N U T, 0, 0, 0',
	X =  176.049  mm,	Y =   -452.328  mm,	Z =   -331.926  mm,
	W =  90.000 deg,	P =   0.000 deg,	R =   90.000 deg
};
P[350]{
   GP1:
	UF : 0, UT : 6,		CONFIG : 'N U T, 0, 0, 0',
	X =  176.672  mm,	Y =   -452.435  mm,	Z =   -329.100  mm,
	W =  90.000 deg,	P =   0.000 deg,	R =   90.000 deg
};
P[351]{
   GP1:
	UF : 0, UT : 6,		CONFIG : 'N U T, 0, 0, 0',
	X =  176.676  mm,	Y =   -451.478  mm,	Z =   -334.185  mm,
	W =  90.000 deg,	P =   0.000 deg,	R =   90.000 deg
};
P[352]{
   GP1:
	UF : 0, UT : 6,		CONFIG : 'N U T, 0, 0, 0',
	X =  177.092  mm,	Y =   -452.141  mm,	Z =   -330.350  mm,
	W =  90.000 deg,	P =   0.000 deg,	R =   90.000 deg
};
P[353]{
   GP1:
	UF : 0, UT : 6,		CONFIG : 'N U T, 0, 0, 0',
	X =  177.117  mm,	Y =   -452.069  mm,	Z =   -330.998  mm,
	W =  90.000 deg,	P =   0.000 deg,	R =   90.000 deg
};
P[354]{
   GP1:
	UF : 0, UT : 6,		CONFIG : 'N U T, 0, 0, 0',
	X =  177.170  mm,	Y =   -451.923  mm,	Z =   -331.928  mm,
	W =  90.000 deg,	P =   0.000 deg,	R =   90.000 deg
};
P[355]{
   GP1:
	UF : 0, UT : 6,		CONFIG : 'N U T, 0, 0, 0',
	X =  177.126  mm,	Y =   -451.700  mm,	Z =   -332.881  mm,
	W =  90.000 deg,	P =   0.000 deg,	R =   90.000 deg
};
P[356]{
   GP1:
	UF : 0, UT : 6,		CONFIG : 'N U T, 0, 0, 0',
	X =  177.776  mm,	Y =   -451.896  mm,	Z =   -330.319  mm,
	W =  90.000 deg,	P =   0.000 deg,	R =   90.000 deg
};
P[357]{
   GP1:
	UF : 0, UT : 6,		CONFIG : 'N U T, 0, 0, 0',
	X =  177.788  mm,	Y =   -451.318  mm,	Z =   -333.402  mm,
	W =  90.000 deg,	P =   0.000 deg,	R =   90.000 deg
};
P[358]{
   GP1:
	UF : 0, UT : 6,		CONFIG : 'N U T, 0, 0, 0',
	X =  178.064  mm,	Y =   -451.597  mm,	Z =   -331.945  mm,
	W =  90.000 deg,	P =   0.000 deg,	R =   90.000 deg
};
P[359]{
   GP1:
	UF : 0, UT : 6,		CONFIG : 'N U T, 0, 0, 0',
	X =  178.071  mm,	Y =   -450.914  mm,	Z =   -334.366  mm,
	W =  90.000 deg,	P =   0.000 deg,	R =   90.000 deg
};
P[360]{
   GP1:
	UF : 0, UT : 6,		CONFIG : 'N U T, 0, 0, 0',
	X =  178.715  mm,	Y =   -450.392  mm,	Z =   -335.089  mm,
	W =  90.000 deg,	P =   0.000 deg,	R =   90.000 deg
};
P[361]{
   GP1:
	UF : 0, UT : 6,		CONFIG : 'N U T, 0, 0, 0',
	X =  179.077  mm,	Y =   -450.919  mm,	Z =   -333.209  mm,
	W =  90.000 deg,	P =   0.000 deg,	R =   90.000 deg
};
P[362]{
   GP1:
	UF : 0, UT : 6,		CONFIG : 'N U T, 0, 0, 0',
	X =  178.996  mm,	Y =   -450.562  mm,	Z =   -334.429  mm,
	W =  90.000 deg,	P =   0.000 deg,	R =   90.000 deg
};
P[363]{
   GP1:
	UF : 0, UT : 6,		CONFIG : 'N U T, 0, 0, 0',
	X =  179.819  mm,	Y =   -450.675  mm,	Z =   -333.142  mm,
	W =  90.000 deg,	P =   0.000 deg,	R =   90.000 deg
};
P[364]{
   GP1:
	UF : 0, UT : 6,		CONFIG : 'N U T, 0, 0, 0',
	X =  179.737  mm,	Y =   -450.416  mm,	Z =   -334.096  mm,
	W =  90.000 deg,	P =   0.000 deg,	R =   90.000 deg
};
P[365]{
   GP1:
	UF : 0, UT : 6,		CONFIG : 'N U T, 0, 0, 0',
	X =  179.631  mm,	Y =   -449.923  mm,	Z =   -335.448  mm,
	W =  90.000 deg,	P =   0.000 deg,	R =   90.000 deg
};
P[366]{
   GP1:
	UF : 0, UT : 6,		CONFIG : 'N U T, 0, 0, 0',
	X =  180.656  mm,	Y =   -450.136  mm,	Z =   -333.957  mm,
	W =  90.000 deg,	P =   0.000 deg,	R =   90.000 deg
};
P[367]{
   GP1:
	UF : 0, UT : 6,		CONFIG : 'N U T, 0, 0, 0',
	X =  180.287  mm,	Y =   -449.485  mm,	Z =   -335.894  mm,
	W =  90.000 deg,	P =   0.000 deg,	R =   90.000 deg
};
P[368]{
   GP1:
	UF : 0, UT : 6,		CONFIG : 'N U T, 0, 0, 0',
	X =  181.130  mm,	Y =   -449.620  mm,	Z =   -334.901  mm,
	W =  90.000 deg,	P =   0.000 deg,	R =   90.000 deg
};
P[369]{
   GP1:
	UF : 0, UT : 6,		CONFIG : 'N U T, 0, 0, 0',
	X =  181.345  mm,	Y =   -449.078  mm,	Z =   -335.986  mm,
	W =  90.000 deg,	P =   0.000 deg,	R =   90.000 deg
};
P[370]{
   GP1:
	UF : 0, UT : 6,		CONFIG : 'N U T, 0, 0, 0',
	X =  181.682  mm,	Y =   -449.618  mm,	Z =   -334.433  mm,
	W =  90.000 deg,	P =   0.000 deg,	R =   90.000 deg
};
P[371]{
   GP1:
	UF : 0, UT : 6,		CONFIG : 'N U T, 0, 0, 0',
	X =  181.911  mm,	Y =   -449.230  mm,	Z =   -335.182  mm,
	W =  90.000 deg,	P =   0.000 deg,	R =   90.000 deg
};
P[372]{
   GP1:
	UF : 0, UT : 6,		CONFIG : 'N U T, 0, 0, 0',
	X =  181.950  mm,	Y =   -448.730  mm,	Z =   -336.262  mm,
	W =  90.000 deg,	P =   0.000 deg,	R =   90.000 deg
};
P[373]{
   GP1:
	UF : 0, UT : 6,		CONFIG : 'N U T, 0, 0, 0',
	X =  182.267  mm,	Y =   -448.289  mm,	Z =   -336.890  mm,
	W =  90.000 deg,	P =   0.000 deg,	R =   90.000 deg
};
P[374]{
   GP1:
	UF : 0, UT : 6,		CONFIG : 'N U T, 0, 0, 0',
	X =  182.857  mm,	Y =   -448.838  mm,	Z =   -335.328  mm,
	W =  90.000 deg,	P =   0.000 deg,	R =   90.000 deg
};
P[375]{
   GP1:
	UF : 0, UT : 6,		CONFIG : 'N U T, 0, 0, 0',
	X =  182.675  mm,	Y =   -448.506  mm,	Z =   -336.218  mm,
	W =  90.000 deg,	P =   0.000 deg,	R =   90.000 deg
};
P[376]{
   GP1:
	UF : 0, UT : 6,		CONFIG : 'N U T, 0, 0, 0',
	X =  183.231  mm,	Y =   -447.995  mm,	Z =   -336.842  mm,
	W =  90.000 deg,	P =   0.000 deg,	R =   90.000 deg
};
P[377]{
   GP1:
	UF : 0, UT : 6,		CONFIG : 'N U T, 0, 0, 0',
	X =  183.649  mm,	Y =   -448.240  mm,	Z =   -336.093  mm,
	W =  90.000 deg,	P =   0.000 deg,	R =   90.000 deg
};
P[378]{
   GP1:
	UF : 0, UT : 6,		CONFIG : 'N U T, 0, 0, 0',
	X =  183.638  mm,	Y =   -447.545  mm,	Z =   -337.366  mm,
	W =  90.000 deg,	P =   0.000 deg,	R =   90.000 deg
};
P[379]{
   GP1:
	UF : 0, UT : 6,		CONFIG : 'N U T, 0, 0, 0',
	X =  184.398  mm,	Y =   -447.303  mm,	Z =   -337.343  mm,
	W =  90.000 deg,	P =   0.000 deg,	R =   90.000 deg
};
P[380]{
   GP1:
	UF : 0, UT : 6,		CONFIG : 'N U T, 0, 0, 0',
	X =  184.974  mm,	Y =   -447.595  mm,	Z =   -336.471  mm,
	W =  90.000 deg,	P =   0.000 deg,	R =   90.000 deg
};
P[381]{
   GP1:
	UF : 0, UT : 6,		CONFIG : 'N U T, 0, 0, 0',
	X =  184.874  mm,	Y =   -446.871  mm,	Z =   -337.800  mm,
	W =  90.000 deg,	P =   0.000 deg,	R =   90.000 deg
};
P[382]{
   GP1:
	UF : 0, UT : 6,		CONFIG : 'N U T, 0, 0, 0',
	X =  185.639  mm,	Y =   -447.103  mm,	Z =   -336.979  mm,
	W =  90.000 deg,	P =   0.000 deg,	R =   90.000 deg
};
P[383]{
   GP1:
	UF : 0, UT : 6,		CONFIG : 'N U T, 0, 0, 0',
	X =  185.453  mm,	Y =   -446.496  mm,	Z =   -338.100  mm,
	W =  90.000 deg,	P =   0.000 deg,	R =   90.000 deg
};
P[384]{
   GP1:
	UF : 0, UT : 6,		CONFIG : 'N U T, 0, 0, 0',
	X =  186.218  mm,	Y =   -446.243  mm,	Z =   -338.093  mm,
	W =  90.000 deg,	P =   0.000 deg,	R =   90.000 deg
};
P[385]{
   GP1:
	UF : 0, UT : 6,		CONFIG : 'N U T, 0, 0, 0',
	X =  186.535  mm,	Y =   -446.517  mm,	Z =   -337.457  mm,
	W =  90.000 deg,	P =   0.000 deg,	R =   90.000 deg
};
P[386]{
   GP1:
	UF : 0, UT : 6,		CONFIG : 'N U T, 0, 0, 0',
	X =  186.388  mm,	Y =   -445.820  mm,	Z =   -338.707  mm,
	W =  90.000 deg,	P =   0.000 deg,	R =   90.000 deg
};
P[387]{
   GP1:
	UF : 0, UT : 6,		CONFIG : 'N U T, 0, 0, 0',
	X =  187.598  mm,	Y =   -445.545  mm,	Z =   -338.487  mm,
	W =  90.000 deg,	P =   0.000 deg,	R =   90.000 deg
};
P[388]{
   GP1:
	UF : 0, UT : 6,		CONFIG : 'N U T, 0, 0, 0',
	X =  188.230  mm,	Y =   -445.731  mm,	Z =   -337.818  mm,
	W =  90.000 deg,	P =   0.000 deg,	R =   90.000 deg
};
P[389]{
   GP1:
	UF : 0, UT : 6,		CONFIG : 'N U T, 0, 0, 0',
	X =  188.367  mm,	Y =   -445.157  mm,	Z =   -338.703  mm,
	W =  90.000 deg,	P =   0.000 deg,	R =   90.000 deg
};
P[390]{
   GP1:
	UF : 0, UT : 6,		CONFIG : 'N U T, 0, 0, 0',
	X =  188.930  mm,	Y =   -444.507  mm,	Z =   -339.389  mm,
	W =  90.000 deg,	P =   0.000 deg,	R =   90.000 deg
};
P[391]{
   GP1:
	UF : 0, UT : 6,		CONFIG : 'N U T, 0, 0, 0',
	X =  189.750  mm,	Y =   -444.885  mm,	Z =   -338.378  mm,
	W =  90.000 deg,	P =   0.000 deg,	R =   90.000 deg
};
P[392]{
   GP1:
	UF : 0, UT : 6,		CONFIG : 'N U T, 0, 0, 0',
	X =  189.549  mm,	Y =   -444.130  mm,	Z =   -339.618  mm,
	W =  90.000 deg,	P =   0.000 deg,	R =   90.000 deg
};
P[393]{
   GP1:
	UF : 0, UT : 6,		CONFIG : 'N U T, 0, 0, 0',
	X =  190.101  mm,	Y =   -444.465  mm,	Z =   -338.887  mm,
	W =  90.000 deg,	P =   0.000 deg,	R =   90.000 deg
};
P[394]{
   GP1:
	UF : 0, UT : 6,		CONFIG : 'N U T, 0, 0, 0',
	X =  190.785  mm,	Y =   -443.938  mm,	Z =   -339.369  mm,
	W =  90.000 deg,	P =   0.000 deg,	R =   90.000 deg
};
P[395]{
   GP1:
	UF : 0, UT : 6,		CONFIG : 'N U T, 0, 0, 0',
	X =  190.685  mm,	Y =   -443.482  mm,	Z =   -339.978  mm,
	W =  90.000 deg,	P =   0.000 deg,	R =   90.000 deg
};
P[396]{
   GP1:
	UF : 0, UT : 6,		CONFIG : 'N U T, 0, 0, 0',
	X =  191.566  mm,	Y =   -443.738  mm,	Z =   -339.278  mm,
	W =  90.000 deg,	P =   0.000 deg,	R =   90.000 deg
};
P[397]{
   GP1:
	UF : 0, UT : 6,		CONFIG : 'N U T, 0, 0, 0',
	X =  191.643  mm,	Y =   -443.065  mm,	Z =   -340.122  mm,
	W =  90.000 deg,	P =   0.000 deg,	R =   90.000 deg
};
P[398]{
   GP1:
	UF : 0, UT : 6,		CONFIG : 'N U T, 0, 0, 0',
	X =  192.520  mm,	Y =   -442.831  mm,	Z =   -340.072  mm,
	W =  90.000 deg,	P =   0.000 deg,	R =   90.000 deg
};
P[399]{
   GP1:
	UF : 0, UT : 6,		CONFIG : 'N U T, 0, 0, 0',
	X =  193.256  mm,	Y =   -442.051  mm,	Z =   -340.748  mm,
	W =  90.000 deg,	P =   0.000 deg,	R =   90.000 deg
};
P[400]{
   GP1:
	UF : 0, UT : 6,		CONFIG : 'N U T, 0, 0, 0',
	X =  193.672  mm,	Y =   -442.580  mm,	Z =   -339.940  mm,
	W =  90.000 deg,	P =   0.000 deg,	R =   90.000 deg
};
P[401]{
   GP1:
	UF : 0, UT : 6,		CONFIG : 'N U T, 0, 0, 0',
	X =  194.058  mm,	Y =   -441.673  mm,	Z =   -340.904  mm,
	W =  90.000 deg,	P =   0.000 deg,	R =   90.000 deg
};
P[402]{
   GP1:
	UF : 0, UT : 6,		CONFIG : 'N U T, 0, 0, 0',
	X =  194.757  mm,	Y =   -441.560  mm,	Z =   -340.716  mm,
	W =  90.000 deg,	P =   0.000 deg,	R =   90.000 deg
};
P[403]{
   GP1:
	UF : 0, UT : 6,		CONFIG : 'N U T, 0, 0, 0',
	X =  195.750  mm,	Y =   -441.354  mm,	Z =   -340.214  mm,
